LIN {X 0,Y 570.27,Z 1282.919,A -85,B 0,C 180,E1 9276.078,E2 9276.078} C_VEL
LIN {X 0,Y 570.578,Z 1274.301,A -85,B 0,C 180,E1 9280.677,E2 9280.677} C_VEL
LIN {X 0,Y 571.345,Z 1260.732,A -85,B 0,C 180,E1 9285.329,E2 9285.329} C_VEL
LIN {X 0,Y 573.008,Z 1241.765,A -85,B 0,C 180,E1 9290.042,E2 9290.042} C_VEL
LIN {X 0,Y 575.848,Z 1217.478,A -85,B 0,C 180,E1 9294.611,E2 9294.611} C_VEL
LIN {X 0,Y 580.222,Z 1187.751,A -85,B 0,C 180,E1 9299.027,E2 9299.027} C_VEL
LIN {X 0,Y 585.818,Z 1152.279,A -85,B 0,C 180,E1 9303.171,E2 9303.171} C_VEL
LIN {X 0,Y 592.121,Z 1114.219,A -85,B 0,C 180,E1 9306.711,E2 9306.711} C_VEL
LIN {X 0,Y 598.707,Z 1072.32,A -85,B 0,C 180,E1 9309.756,E2 9309.756} C_VEL
LIN {X 0,Y 603.11,Z 1037.935,A -85,B 0,C 180,E1 9311.685,E2 9311.685} C_VEL
LIN {X 0,Y 607.858,Z 987.119,A -85,B 0,C 180,E1 9313.723,E2 9313.723} C_VEL
LIN {X 0,Y 611.73,Z 933.476,A -85,B 0,C 180,E1 9315.186,E2 9315.186} C_VEL
LIN {X 0,Y 613.598,Z 886.911,A -85,B 0,C 180,E1 9315.996,E2 9315.996} C_VEL
LIN {X 0,Y 590.85,Z 850.721,A -85,B 0,C 180,E1 9318.163,E2 9318.163} C_VEL
LIN {X 0,Y 571.274,Z 814.347,A -85,B 0,C 180,E1 9320.427,E2 9320.427} C_VEL
LIN {X 0,Y 569.24,Z 809.06,A -85,B 0,C 180,E1 9320.777,E2 9320.777} C_VEL
LIN {X 0,Y 569.158,Z 809.06,A -85,B 0,C 180,E1 9326.116,E2 9326.116} C_VEL
LIN {X 0,Y 569.253,Z 809.06,A -85,B 0,C 180,E1 9331.459,E2 9331.459} C_VEL
LIN {X 0,Y 569.293,Z 809.111,A -85,B 0,C 180,E1 9336.25,E2 9336.25} C_VEL
LIN {X 0,Y 571.892,Z 814.911,A -85,B 0,C 180,E1 9336.731,E2 9336.731} C_VEL
LIN {X 0,Y 590.013,Z 852.89,A -85,B 0,C 180,E1 9340.042,E2 9340.042} C_VEL
LIN {X 0,Y 603.31,Z 886.116,A -85,B 0,C 180,E1 9343.049,E2 9343.049} C_VEL
LIN {X 0,Y 601.143,Z 906.53,A -85,B 0,C 180,E1 9344.23,E2 9344.23} C_VEL
LIN {X 0,Y 594.464,Z 949.147,A -85,B 0,C 180,E1 9347.056,E2 9347.056} C_VEL
LIN {X 0,Y 588.168,Z 988.3,A -85,B 0,C 180,E1 9350.387,E2 9350.387} C_VEL
LIN {X 0,Y 582.328,Z 1024.228,A -85,B 0,C 180,E1 9354.229,E2 9354.229} C_VEL
LIN {X 0,Y 577.319,Z 1057.198,A -85,B 0,C 180,E1 9358.687,E2 9358.687} C_VEL
LIN {X 0,Y 573.896,Z 1084.316,A -85,B 0,C 180,E1 9363.396,E2 9363.396} C_VEL
LIN {X 0,Y 571.748,Z 1105.972,A -85,B 0,C 180,E1 9368.299,E2 9368.299} C_VEL
LIN {X 0,Y 570.726,Z 1121.122,A -85,B 0,C 180,E1 9373.004,E2 9373.004} C_VEL
LIN {X 0,Y 570.222,Z 1130.776,A -85,B 0,C 180,E1 9377.472,E2 9377.472} C_VEL
LIN {X 0,Y 569.748,Z 1135.899,A -85,B 0,C 180,E1 9381.854,E2 9381.854} C_VEL
LIN {X 0,Y 569.684,Z 1136.615,A -85,B 0,C 180,E1 9386.801,E2 9386.801} C_VEL
LIN {X 0,Y 570.107,Z 1133.109,A -85,B 0,C 180,E1 9390.855,E2 9390.855} C_VEL
LIN {X 0,Y 570.541,Z 1124.317,A -85,B 0,C 180,E1 9395.635,E2 9395.635} C_VEL
LIN {X 0,Y 571.308,Z 1110.925,A -85,B 0,C 180,E1 9400.236,E2 9400.236} C_VEL
LIN {X 0,Y 572.975,Z 1091.952,A -85,B 0,C 180,E1 9404.949,E2 9404.949} C_VEL
LIN {X 0,Y 575.904,Z 1067.652,A -85,B 0,C 180,E1 9409.54,E2 9409.54} C_VEL
LIN {X 0,Y 580.109,Z 1037.955,A -85,B 0,C 180,E1 9413.951,E2 9413.951} C_VEL
LIN {X 0,Y 585.487,Z 1004.176,A -85,B 0,C 180,E1 9417.936,E2 9417.936} C_VEL
LIN {X 0,Y 591.862,Z 965.664,A -85,B 0,C 180,E1 9421.545,E2 9421.545} C_VEL
LIN {X 0,Y 598.661,Z 923.01,A -85,B 0,C 180,E1 9424.677,E2 9424.677} C_VEL
LIN {X 0,Y 603.556,Z 886.886,A -85,B 0,C 180,E1 9426.783,E2 9426.783} C_VEL
LIN {X 0,Y 589.393,Z 850.595,A -85,B 0,C 180,E1 9430.148,E2 9430.148} C_VEL
LIN {X 0,Y 571.501,Z 814.431,A -85,B 0,C 180,E1 9433.642,E2 9433.642} C_VEL
LIN {X 0,Y 569.436,Z 809.06,A -85,B 0,C 180,E1 9434.125,E2 9434.125} C_VEL
LIN {X 0,Y 569.824,Z 809.06,A -85,B 0,C 180,E1 9439.309,E2 9439.309} C_VEL
LIN {X 0,Y 570.01,Z 809.06,A -85,B 0,C 180,E1 9443.919,E2 9443.919} C_VEL
LIN {X 0,Y 570.065,Z 809.06,A -85,B 0,C 180,E1 9448.487,E2 9448.487} C_VEL
LIN {X 0,Y 570.001,Z 809.06,A -85,B 0,C 180,E1 9453.045,E2 9453.045} C_VEL
LIN {X 0,Y 569.951,Z 809.06,A -85,B 0,C 180,E1 9457.624,E2 9457.624} C_VEL
LIN {X 0,Y 569.806,Z 809.06,A -85,B 0,C 180,E1 9462.255,E2 9462.255} C_VEL
LIN {X 0,Y 569.672,Z 809.06,A -85,B 0,C 180,E1 9467.283,E2 9467.283} C_VEL
LIN {X 0,Y 569.54,Z 809.06,A -85,B 0,C 180,E1 9471.811,E2 9471.811} C_VEL
LIN {X 0,Y 569.423,Z 809.06,A -85,B 0,C 180,E1 9476.822,E2 9476.822} C_VEL
LIN {X 0,Y 569.313,Z 809.06,A -85,B 0,C 180,E1 9482.069,E2 9482.069} C_VEL
LIN {X 0,Y 569.252,Z 809.06,A -85,B 0,C 180,E1 9487.635,E2 9487.635} C_VEL
LIN {X 0,Y 569.19,Z 809.06,A -85,B 0,C 180,E1 9493.657,E2 9493.657} C_VEL
LIN {X 0,Y 569.157,Z 809.06,A -85,B 0,C 180,E1 9498.418,E2 9498.418} C_VEL
LIN {X 0,Y 569.22,Z 809.06,A -85,B 0,C 180,E1 9504.269,E2 9504.269} C_VEL
LIN {X 0,Y 569.324,Z 809.06,A -85,B 0,C 180,E1 9509.718,E2 9509.718} C_VEL
LIN {X 0,Y 569.49,Z 809.06,A -85,B 0,C 180,E1 9514.881,E2 9514.881} C_VEL
LIN {X 0,Y 569.623,Z 809.06,A -85,B 0,C 180,E1 9519.829,E2 9519.829} C_VEL
LIN {X 0,Y 569.678,Z 809.06,A -85,B 0,C 180,E1 9524.62,E2 9524.62} C_VEL
LIN {X 0,Y 569.836,Z 809.06,A -85,B 0,C 180,E1 9529.304,E2 9529.304} C_VEL
LIN {X 0,Y 570.009,Z 809.06,A -85,B 0,C 180,E1 9533.914,E2 9533.914} C_VEL
LIN {X 0,Y 570.293,Z 809.06,A -85,B 0,C 180,E1 9540.001,E2 9540.001} C_VEL
LIN {X 0,Y 570.05,Z 809.06,A -85,B 0,C 180,E1 9546.087,E2 9546.087} C_VEL
LIN {X 0,Y 569.806,Z 809.06,A -85,B 0,C 180,E1 9552.248,E2 9552.248} C_VEL
LIN {X 0,Y 569.663,Z 809.06,A -85,B 0,C 180,E1 9557.251,E2 9557.251} C_VEL
LIN {X 0,Y 569.537,Z 809.06,A -85,B 0,C 180,E1 9561.804,E2 9561.804} C_VEL
LIN {X 0,Y 569.373,Z 809.06,A -85,B 0,C 180,E1 9566.818,E2 9566.818} C_VEL
LIN {X 0,Y 569.312,Z 809.06,A -85,B 0,C 180,E1 9572.061,E2 9572.061} C_VEL
LIN {X 0,Y 569.281,Z 809.538,A -85,B 0,C 180,E1 9577.816,E2 9577.816} C_VEL
LIN {X 0,Y 571.948,Z 814.98,A -85,B 0,C 180,E1 9578.222,E2 9578.222} C_VEL
LIN {X 0,Y 598.675,Z 858.988,A -85,B 0,C 180,E1 9581.795,E2 9581.795} C_VEL
LIN {X 0,Y 615.701,Z 888.66,A -85,B 0,C 180,E1 9583.807,E2 9583.807} C_VEL
LIN {X 0,Y 613.152,Z 939.54,A -85,B 0,C 180,E1 9584.758,E2 9584.758} C_VEL
LIN {X 0,Y 609.127,Z 984.504,A -85,B 0,C 180,E1 9586.049,E2 9586.049} C_VEL
LIN {X 0,Y 604.919,Z 1025.197,A -85,B 0,C 180,E1 9587.692,E2 9587.692} C_VEL
LIN {X 0,Y 599.652,Z 1040.997,A -85,B 0,C 180,E1 9588.224,E2 9588.224} C_VEL
LIN {X 0,Y 594.647,Z 1054.535,A -85,B 0,C 180,E1 9588.734,E2 9588.734} C_VEL
LIN {X 0,Y 594.367,Z 1056.402,A -85,B 0,C 180,E1 9588.836,E2 9588.836} C_VEL
LIN {X 0,Y 589.081,Z 1093.061,A -85,B 0,C 180,E1 9591.166,E2 9591.166} C_VEL
LIN {X 0,Y 582.379,Z 1132.494,A -85,B 0,C 180,E1 9594.416,E2 9594.416} C_VEL
LIN {X 0,Y 575.672,Z 1171.448,A -85,B 0,C 180,E1 9598.523,E2 9598.523} C_VEL
LIN {X 0,Y 570.444,Z 1203.465,A -85,B 0,C 180,E1 9602.806,E2 9602.806} C_VEL
LIN {X 0,Y 566.697,Z 1230.555,A -85,B 0,C 180,E1 9607.393,E2 9607.393} C_VEL
LIN {X 0,Y 564.414,Z 1251.77,A -85,B 0,C 180,E1 9612.025,E2 9612.025} C_VEL
LIN {X 0,Y 562.989,Z 1268.116,A -85,B 0,C 180,E1 9616.806,E2 9616.806} C_VEL
LIN {X 0,Y 562.467,Z 1279.21,A -85,B 0,C 180,E1 9621.497,E2 9621.497} C_VEL
LIN {X 0,Y 562.279,Z 1284.659,A -85,B 0,C 180,E1 9625.369,E2 9625.369} C_VEL
LIN {X 0,Y 562.346,Z 1287,A -85,B 0,C 180,E1 9629.994,E2 9629.994} C_VEL
LIN {X 0,Y 562.279,Z 1284.673,A -85,B 0,C 180,E1 9634.618,E2 9634.618} C_VEL
LIN {X 0,Y 562.448,Z 1277.69,A -85,B 0,C 180,E1 9639.27,E2 9639.27} C_VEL
LIN {X 0,Y 563.222,Z 1265.86,A -85,B 0,C 180,E1 9643.966,E2 9643.966} C_VEL
LIN {X 0,Y 564.723,Z 1248.729,A -85,B 0,C 180,E1 9648.722,E2 9648.722} C_VEL
LIN {X 0,Y 567.547,Z 1224.45,A -85,B 0,C 180,E1 9653.74,E2 9653.74} C_VEL
LIN {X 0,Y 571.579,Z 1196.601,A -85,B 0,C 180,E1 9658.197,E2 9658.197} C_VEL
LIN {X 0,Y 577.41,Z 1161.259,A -85,B 0,C 180,E1 9662.659,E2 9662.659} C_VEL
LIN {X 0,Y 583.923,Z 1123.342,A -85,B 0,C 180,E1 9666.403,E2 9666.403} C_VEL
LIN {X 0,Y 590.741,Z 1082.843,A -85,B 0,C 180,E1 9669.569,E2 9669.569} C_VEL
LIN {X 0,Y 595.524,Z 1043.572,A -85,B 0,C 180,E1 9671.766,E2 9671.766} C_VEL
LIN {X 0,Y 600.653,Z 991.518,A -85,B 0,C 180,E1 9673.943,E2 9673.943} C_VEL
LIN {X 0,Y 604.673,Z 940.832,A -85,B 0,C 180,E1 9675.437,E2 9675.437} C_VEL
LIN {X 0,Y 607.027,Z 889.973,A -85,B 0,C 180,E1 9676.388,E2 9676.388} C_VEL
LIN {X 0,Y 585.603,Z 855.505,A -85,B 0,C 180,E1 9678.501,E2 9678.501} C_VEL
LIN {X 0,Y 566.705,Z 819.88,A -85,B 0,C 180,E1 9680.764,E2 9680.764} C_VEL
LIN {X 0,Y 561.456,Z 810.557,A -85,B 0,C 180,E1 9681.473,E2 9681.473} C_VEL
LIN {X 0,Y 561.314,Z 809.06,A -85,B 0,C 180,E1 9681.557,E2 9681.557} C_VEL
LIN {X 0,Y 561.235,Z 809.06,A -85,B 0,C 180,E1 9687.421,E2 9687.421} C_VEL
LIN {X 0,Y 561.342,Z 809.06,A -85,B 0,C 180,E1 9692.767,E2 9692.767} C_VEL
LIN {X 0,Y 561.39,Z 809.624,A -85,B 0,C 180,E1 9695.4,E2 9695.4} C_VEL
LIN {X 0,Y 567.085,Z 820.612,A -85,B 0,C 180,E1 9696.428,E2 9696.428} C_VEL
LIN {X 0,Y 584.99,Z 858.969,A -85,B 0,C 180,E1 9699.894,E2 9699.894} C_VEL
LIN {X 0,Y 597.178,Z 890.245,A -85,B 0,C 180,E1 9702.783,E2 9702.783} C_VEL
LIN {X 0,Y 590.812,Z 932.783,A -85,B 0,C 180,E1 9705.371,E2 9705.371} C_VEL
LIN {X 0,Y 583.573,Z 975.191,A -85,B 0,C 180,E1 9708.707,E2 9708.707} C_VEL
LIN {X 0,Y 577.139,Z 1012.847,A -85,B 0,C 180,E1 9712.478,E2 9712.478} C_VEL
LIN {X 0,Y 571.505,Z 1046.855,A -85,B 0,C 180,E1 9716.779,E2 9716.779} C_VEL
LIN {X 0,Y 567.399,Z 1075.144,A -85,B 0,C 180,E1 9721.335,E2 9721.335} C_VEL
LIN {X 0,Y 564.565,Z 1098.396,A -85,B 0,C 180,E1 9726.145,E2 9726.145} C_VEL
LIN {X 0,Y 563.206,Z 1115.371,A -85,B 0,C 180,E1 9730.824,E2 9730.824} C_VEL
LIN {X 0,Y 562.453,Z 1127.522,A -85,B 0,C 180,E1 9735.583,E2 9735.583} C_VEL
LIN {X 0,Y 562.058,Z 1134.141,A -85,B 0,C 180,E1 9739.808,E2 9739.808} C_VEL
LIN {X 0,Y 561.734,Z 1136.813,A -85,B 0,C 180,E1 9743.868,E2 9743.868} C_VEL
LIN {X 0,Y 561.918,Z 1135.246,A -85,B 0,C 180,E1 9748.947,E2 9748.947} C_VEL
LIN {X 0,Y 562.493,Z 1128.891,A -85,B 0,C 180,E1 9753.628,E2 9753.628} C_VEL
LIN {X 0,Y 563.215,Z 1117.089,A -85,B 0,C 180,E1 9758.519,E2 9758.519} C_VEL
LIN {X 0,Y 564.477,Z 1099.987,A -85,B 0,C 180,E1 9763.383,E2 9763.383} C_VEL
LIN {X 0,Y 566.914,Z 1078.804,A -85,B 0,C 180,E1 9767.898,E2 9767.898} C_VEL
LIN {X 0,Y 570.861,Z 1050.717,A -85,B 0,C 180,E1 9772.565,E2 9772.565} C_VEL
LIN {X 0,Y 576.205,Z 1017.971,A -85,B 0,C 180,E1 9776.844,E2 9776.844} C_VEL
LIN {X 0,Y 582.483,Z 981.653,A -85,B 0,C 180,E1 9780.615,E2 9780.615} C_VEL
LIN {X 0,Y 589.351,Z 941.758,A -85,B 0,C 180,E1 9783.889,E2 9783.889} C_VEL
LIN {X 0,Y 595.881,Z 900.345,A -85,B 0,C 180,E1 9786.563,E2 9786.563} C_VEL
LIN {X 0,Y 597.083,Z 889.866,A -85,B 0,C 180,E1 9787.156,E2 9787.156} C_VEL
LIN {X 0,Y 583.392,Z 854.423,A -85,B 0,C 180,E1 9790.527,E2 9790.527} C_VEL
LIN {X 0,Y 566.082,Z 819.268,A -85,B 0,C 180,E1 9794.026,E2 9794.026} C_VEL
LIN {X 0,Y 561.565,Z 809.06,A -85,B 0,C 180,E1 9795.024,E2 9795.024} C_VEL
LIN {X 0,Y 561.986,Z 809.06,A -85,B 0,C 180,E1 9800.723,E2 9800.723} C_VEL
LIN {X 0,Y 562.129,Z 809.06,A -85,B 0,C 180,E1 9805.381,E2 9805.381} C_VEL
LIN {X 0,Y 562.245,Z 809.06,A -85,B 0,C 180,E1 9811.546,E2 9811.546} C_VEL
LIN {X 0,Y 562.11,Z 809.06,A -85,B 0,C 180,E1 9816.179,E2 9816.179} C_VEL
LIN {X 0,Y 561.94,Z 809.06,A -85,B 0,C 180,E1 9820.856,E2 9820.856} C_VEL
LIN {X 0,Y 561.813,Z 809.06,A -85,B 0,C 180,E1 9825.609,E2 9825.609} C_VEL
LIN {X 0,Y 561.669,Z 809.06,A -85,B 0,C 180,E1 9830.478,E2 9830.478} C_VEL
LIN {X 0,Y 561.519,Z 809.06,A -85,B 0,C 180,E1 9835.51,E2 9835.51} C_VEL
LIN {X 0,Y 561.41,Z 809.06,A -85,B 0,C 180,E1 9840.764,E2 9840.764} C_VEL
LIN {X 0,Y 561.34,Z 809.06,A -85,B 0,C 180,E1 9846.322,E2 9846.322} C_VEL
LIN {X 0,Y 561.249,Z 809.06,A -85,B 0,C 180,E1 9852.313,E2 9852.313} C_VEL
LIN {X 0,Y 561.215,Z 809.06,A -85,B 0,C 180,E1 9857.695,E2 9857.695} C_VEL
LIN {X 0,Y 561.288,Z 809.06,A -85,B 0,C 180,E1 9863.876,E2 9863.876} C_VEL
LIN {X 0,Y 561.394,Z 809.06,A -85,B 0,C 180,E1 9869.476,E2 9869.476} C_VEL
LIN {X 0,Y 561.589,Z 809.06,A -85,B 0,C 180,E1 9874.502,E2 9874.502} C_VEL
LIN {X 0,Y 561.707,Z 809.06,A -85,B 0,C 180,E1 9880.329,E2 9880.329} C_VEL
LIN {X 0,Y 561.779,Z 809.06,A -85,B 0,C 180,E1 9885.992,E2 9885.992} C_VEL
LIN {X 0,Y 562.015,Z 809.06,A -85,B 0,C 180,E1 9890.718,E2 9890.718} C_VEL
LIN {X 0,Y 562.162,Z 809.06,A -85,B 0,C 180,E1 9895.376,E2 9895.376} C_VEL
LIN {X 0,Y 562.382,Z 809.06,A -85,B 0,C 180,E1 9901.54,E2 9901.54} C_VEL
LIN {X 0,Y 562.143,Z 809.06,A -85,B 0,C 180,E1 9906.173,E2 9906.173} C_VEL
LIN {X 0,Y 561.943,Z 809.06,A -85,B 0,C 180,E1 9910.85,E2 9910.85} C_VEL
LIN {X 0,Y 561.789,Z 809.06,A -85,B 0,C 180,E1 9915.603,E2 9915.603} C_VEL
LIN {X 0,Y 561.66,Z 809.06,A -85,B 0,C 180,E1 9920.471,E2 9920.471} C_VEL
LIN {X 0,Y 561.494,Z 809.06,A -85,B 0,C 180,E1 9925.504,E2 9925.504} C_VEL
LIN {X 0,Y 561.401,Z 809.06,A -85,B 0,C 180,E1 9930.756,E2 9930.756} C_VEL
LIN {X 0,Y 561.363,Z 809.06,A -85,B 0,C 180,E1 9936.9,E2 9936.9} C_VEL
LIN {X 0,Y 563.774,Z 814.722,A -85,B 0,C 180,E1 9937.305,E2 9937.305} C_VEL
LIN {X 0,Y 591.925,Z 860.297,A -85,B 0,C 180,E1 9941.157,E2 9941.157} C_VEL
LIN {X 0,Y 609.778,Z 892.169,A -85,B 0,C 180,E1 9943.358,E2 9943.358} C_VEL
LIN {X 0,Y 606.664,Z 945.689,A -85,B 0,C 180,E1 9944.411,E2 9944.411} C_VEL
LIN {X 0,Y 602.242,Z 991.336,A -85,B 0,C 180,E1 9945.821,E2 9945.821} C_VEL
LIN {X 0,Y 596.519,Z 1040.194,A -85,B 0,C 180,E1 9947.969,E2 9947.969} C_VEL
LIN {X 0,Y 594.367,Z 1056.402,A -85,B 0,C 180,E1 9948.836,E2 9948.836} C_VEL
LIN {X 0,Y 590.876,Z 1067.886,A -85,B 0,C 180,E1 9949.369,E2 9949.369} C_VEL
LIN {X 0,Y 583.812,Z 1084.601,A -85,B 0,C 180,E1 9950.139,E2 9950.139} C_VEL
LIN {X 0,Y 583.429,Z 1086.38,A -85,B 0,C 180,E1 9950.256,E2 9950.256} C_VEL
LIN {X 0,Y 577.779,Z 1120.685,A -85,B 0,C 180,E1 9952.876,E2 9952.876} C_VEL
LIN {X 0,Y 570.593,Z 1160.391,A -85,B 0,C 180,E1 9956.791,E2 9956.791} C_VEL
LIN {X 0,Y 564.417,Z 1195.079,A -85,B 0,C 180,E1 9961.184,E2 9961.184} C_VEL
LIN {X 0,Y 560.043,Z 1223.282,A -85,B 0,C 180,E1 9965.697,E2 9965.697} C_VEL
LIN {X 0,Y 557.015,Z 1246.941,A -85,B 0,C 180,E1 9970.584,E2 9970.584} C_VEL
LIN {X 0,Y 555.479,Z 1264.335,A -85,B 0,C 180,E1 9975.314,E2 9975.314} C_VEL
LIN {X 0,Y 554.708,Z 1276.093,A -85,B 0,C 180,E1 9979.795,E2 9979.795} C_VEL
LIN {X 0,Y 554.545,Z 1282.902,A -85,B 0,C 180,E1 9983.736,E2 9983.736} C_VEL
LIN {X 0,Y 554.354,Z 1286.665,A -85,B 0,C 180,E1 9988.432,E2 9988.432} C_VEL
LIN {X 0,Y 554.494,Z 1285.879,A -85,B 0,C 180,E1 9993.118,E2 9993.118} C_VEL
LIN {X 0,Y 554.505,Z 1280.558,A -85,B 0,C 180,E1 9997.825,E2 9997.825} C_VEL
LIN {X 0,Y 555.052,Z 1270.437,A -85,B 0,C 180,E1 10002.573,E2 10002.573} C_VEL
LIN {X 0,Y 556.257,Z 1255.027,A -85,B 0,C 180,E1 10007.379,E2 10007.379} C_VEL
LIN {X 0,Y 558.828,Z 1232.701,A -85,B 0,C 180,E1 10012.516,E2 10012.516} C_VEL
LIN {X 0,Y 562.749,Z 1206.183,A -85,B 0,C 180,E1 10017.152,E2 10017.152} C_VEL
LIN {X 0,Y 568.149,Z 1174.436,A -85,B 0,C 180,E1 10021.556,E2 10021.556} C_VEL
LIN {X 0,Y 574.679,Z 1137.631,A -85,B 0,C 180,E1 10025.566,E2 10025.566} C_VEL
LIN {X 0,Y 581.17,Z 1100.835,A -85,B 0,C 180,E1 10028.741,E2 10028.741} C_VEL
LIN {X 0,Y 586.709,Z 1058.959,A -85,B 0,C 180,E1 10031.311,E2 10031.311} C_VEL
LIN {X 0,Y 592.045,Z 1011.546,A -85,B 0,C 180,E1 10033.551,E2 10033.551} C_VEL
LIN {X 0,Y 596.302,Z 965.395,A -85,B 0,C 180,E1 10035.188,E2 10035.188} C_VEL
LIN {X 0,Y 599.852,Z 915.853,A -85,B 0,C 180,E1 10036.375,E2 10036.375} C_VEL
LIN {X 0,Y 600.289,Z 892.715,A -85,B 0,C 180,E1 10036.808,E2 10036.808} C_VEL
LIN {X 0,Y 580.66,Z 860.751,A -85,B 0,C 180,E1 10038.818,E2 10038.818} C_VEL
LIN {X 0,Y 561.82,Z 824.949,A -85,B 0,C 180,E1 10041.155,E2 10041.155} C_VEL
LIN {X 0,Y 553.395,Z 809.959,A -85,B 0,C 180,E1 10042.379,E2 10042.379} C_VEL
LIN {X 0,Y 553.322,Z 809.06,A -85,B 0,C 180,E1 10042.664,E2 10042.664} C_VEL
LIN {X 0,Y 553.335,Z 809.06,A -85,B 0,C 180,E1 10048.745,E2 10048.745} C_VEL
LIN {X 0,Y 553.505,Z 809.41,A -85,B 0,C 180,E1 10054.458,E2 10054.458} C_VEL
LIN {X 0,Y 556.013,Z 814.843,A -85,B 0,C 180,E1 10054.944,E2 10054.944} C_VEL
LIN {X 0,Y 572.142,Z 846.836,A -85,B 0,C 180,E1 10058.053,E2 10058.053} C_VEL
LIN {X 0,Y 588.015,Z 885.193,A -85,B 0,C 180,E1 10061.64,E2 10061.64} C_VEL
LIN {X 0,Y 590.789,Z 895.257,A -85,B 0,C 180,E1 10062.545,E2 10062.545} C_VEL
LIN {X 0,Y 584.32,Z 935.414,A -85,B 0,C 180,E1 10065.013,E2 10065.013} C_VEL
LIN {X 0,Y 576.622,Z 976.931,A -85,B 0,C 180,E1 10068.378,E2 10068.378} C_VEL
LIN {X 0,Y 569.917,Z 1014.273,A -85,B 0,C 180,E1 10072.19,E2 10072.19} C_VEL
LIN {X 0,Y 564.035,Z 1047.94,A -85,B 0,C 180,E1 10076.544,E2 10076.544} C_VEL
LIN {X 0,Y 559.732,Z 1076.008,A -85,B 0,C 180,E1 10081.16,E2 10081.16} C_VEL
LIN {X 0,Y 556.861,Z 1098.253,A -85,B 0,C 180,E1 10085.84,E2 10085.84} C_VEL
LIN {X 0,Y 555.383,Z 1115.255,A -85,B 0,C 180,E1 10090.581,E2 10090.581} C_VEL
LIN {X 0,Y 554.621,Z 1126.648,A -85,B 0,C 180,E1 10095.007,E2 10095.007} C_VEL
LIN {X 0,Y 554.269,Z 1133.364,A -85,B 0,C 180,E1 10099.094,E2 10099.094} C_VEL
LIN {X 0,Y 553.879,Z 1136.295,A -85,B 0,C 180,E1 10102.452,E2 10102.452} C_VEL
LIN {X 0,Y 553.875,Z 1136.202,A -85,B 0,C 180,E1 10107.63,E2 10107.63} C_VEL
LIN {X 0,Y 554.431,Z 1131.238,A -85,B 0,C 180,E1 10112.354,E2 10112.354} C_VEL
LIN {X 0,Y 554.941,Z 1122.283,A -85,B 0,C 180,E1 10116.799,E2 10116.799} C_VEL
LIN {X 0,Y 556.067,Z 1107.32,A -85,B 0,C 180,E1 10121.734,E2 10121.734} C_VEL
LIN {X 0,Y 558.561,Z 1085.383,A -85,B 0,C 180,E1 10126.918,E2 10126.918} C_VEL
LIN {X 0,Y 562.225,Z 1059.784,A -85,B 0,C 180,E1 10131.546,E2 10131.546} C_VEL
LIN {X 0,Y 567.33,Z 1028.5,A -85,B 0,C 180,E1 10135.999,E2 10135.999} C_VEL
LIN {X 0,Y 573.689,Z 993.193,A -85,B 0,C 180,E1 10139.978,E2 10139.978} C_VEL
LIN {X 0,Y 581.167,Z 952.357,A -85,B 0,C 180,E1 10143.61,E2 10143.61} C_VEL
LIN {X 0,Y 588.328,Z 909.971,A -85,B 0,C 180,E1 10146.541,E2 10146.541} C_VEL
LIN {X 0,Y 590.888,Z 893.797,A -85,B 0,C 180,E1 10147.45,E2 10147.45} C_VEL
LIN {X 0,Y 577.472,Z 858.329,A -85,B 0,C 180,E1 10150.903,E2 10150.903} C_VEL
LIN {X 0,Y 559.287,Z 820.62,A -85,B 0,C 180,E1 10154.734,E2 10154.734} C_VEL
LIN {X 0,Y 553.858,Z 810.471,A -85,B 0,C 180,E1 10155.793,E2 10155.793} C_VEL
LIN {X 0,Y 553.777,Z 809.06,A -85,B 0,C 180,E1 10155.992,E2 10155.992} C_VEL
LIN {X 0,Y 554.063,Z 809.06,A -85,B 0,C 180,E1 10160.589,E2 10160.589} C_VEL
LIN {X 0,Y 554.252,Z 809.06,A -85,B 0,C 180,E1 10165.315,E2 10165.315} C_VEL
LIN {X 0,Y 554.346,Z 809.06,A -85,B 0,C 180,E1 10171.568,E2 10171.568} C_VEL
LIN {X 0,Y 554.195,Z 809.06,A -85,B 0,C 180,E1 10176.268,E2 10176.268} C_VEL
LIN {X 0,Y 554.027,Z 809.06,A -85,B 0,C 180,E1 10181.013,E2 10181.013} C_VEL
LIN {X 0,Y 553.884,Z 809.06,A -85,B 0,C 180,E1 10185.838,E2 10185.838} C_VEL
LIN {X 0,Y 553.719,Z 809.06,A -85,B 0,C 180,E1 10190.785,E2 10190.785} C_VEL
LIN {X 0,Y 553.572,Z 809.06,A -85,B 0,C 180,E1 10195.903,E2 10195.903} C_VEL
LIN {X 0,Y 553.436,Z 809.06,A -85,B 0,C 180,E1 10201.256,E2 10201.256} C_VEL
LIN {X 0,Y 553.346,Z 809.06,A -85,B 0,C 180,E1 10206.933,E2 10206.933} C_VEL
LIN {X 0,Y 553.361,Z 809.06,A -85,B 0,C 180,E1 10213.061,E2 10213.061} C_VEL
LIN {X 0,Y 553.29,Z 809.06,A -85,B 0,C 180,E1 10219.049,E2 10219.049} C_VEL
LIN {X 0,Y 553.348,Z 809.06,A -85,B 0,C 180,E1 10225.018,E2 10225.018} C_VEL
LIN {X 0,Y 553.55,Z 809.06,A -85,B 0,C 180,E1 10230.883,E2 10230.883} C_VEL
LIN {X 0,Y 553.643,Z 809.06,A -85,B 0,C 180,E1 10235.835,E2 10235.835} C_VEL
LIN {X 0,Y 553.835,Z 809.06,A -85,B 0,C 180,E1 10240.89,E2 10240.89} C_VEL
LIN {X 0,Y 553.883,Z 809.06,A -85,B 0,C 180,E1 10245.788,E2 10245.788} C_VEL
LIN {X 0,Y 554.091,Z 809.06,A -85,B 0,C 180,E1 10250.584,E2 10250.584} C_VEL
LIN {X 0,Y 554.262,Z 809.06,A -85,B 0,C 180,E1 10255.309,E2 10255.309} C_VEL
LIN {X 0,Y 554.478,Z 809.06,A -85,B 0,C 180,E1 10261.562,E2 10261.562} C_VEL
LIN {X 0,Y 554.227,Z 809.06,A -85,B 0,C 180,E1 10266.261,E2 10266.261} C_VEL
LIN {X 0,Y 554.021,Z 809.06,A -85,B 0,C 180,E1 10271.007,E2 10271.007} C_VEL
LIN {X 0,Y 553.861,Z 809.06,A -85,B 0,C 180,E1 10277.258,E2 10277.258} C_VEL
LIN {X 0,Y 553.63,Z 809.06,A -85,B 0,C 180,E1 10282.464,E2 10282.464} C_VEL
LIN {X 0,Y 553.504,Z 809.06,A -85,B 0,C 180,E1 10287.651,E2 10287.651} C_VEL
LIN {X 0,Y 553.421,Z 809.06,A -85,B 0,C 180,E1 10293.097,E2 10293.097} C_VEL
LIN {X 0,Y 553.462,Z 809.06,A -85,B 0,C 180,E1 10295.952,E2 10295.952} C_VEL
LIN {X 0,Y 555.857,Z 814.736,A -85,B 0,C 180,E1 10296.375,E2 10296.375} C_VEL
LIN {X 0,Y 585.368,Z 861.947,A -85,B 0,C 180,E1 10300.526,E2 10300.526} C_VEL
LIN {X 0,Y 603.778,Z 894.099,A -85,B 0,C 180,E1 10302.863,E2 10302.863} C_VEL
LIN {X 0,Y 600.627,Z 946.855,A -85,B 0,C 180,E1 10303.942,E2 10303.942} C_VEL
LIN {X 0,Y 595.992,Z 991.688,A -85,B 0,C 180,E1 10305.357,E2 10305.357} C_VEL
LIN {X 0,Y 589.933,Z 1040.905,A -85,B 0,C 180,E1 10307.552,E2 10307.552} C_VEL
LIN {X 0,Y 583.429,Z 1086.38,A -85,B 0,C 180,E1 10310.256,E2 10310.256} C_VEL
LIN {X 0,Y 577.747,Z 1100.839,A -85,B 0,C 180,E1 10311.06,E2 10311.06} C_VEL
LIN {X 0,Y 572.077,Z 1114.879,A -85,B 0,C 180,E1 10311.934,E2 10311.934} C_VEL
LIN {X 0,Y 566.629,Z 1145.24,A -85,B 0,C 180,E1 10314.703,E2 10314.703} C_VEL
LIN {X 0,Y 559.854,Z 1180.913,A -85,B 0,C 180,E1 10318.84,E2 10318.84} C_VEL
LIN {X 0,Y 554.546,Z 1211.371,A -85,B 0,C 180,E1 10323.275,E2 10323.275} C_VEL
LIN {X 0,Y 550.48,Z 1237.847,A -85,B 0,C 180,E1 10328.242,E2 10328.242} C_VEL
LIN {X 0,Y 548.2,Z 1257.996,A -85,B 0,C 180,E1 10333.17,E2 10333.17} C_VEL
LIN {X 0,Y 546.996,Z 1272.347,A -85,B 0,C 180,E1 10338.036,E2 10338.036} C_VEL
LIN {X 0,Y 546.644,Z 1281.741,A -85,B 0,C 180,E1 10342.848,E2 10342.848} C_VEL
LIN {X 0,Y 546.536,Z 1285.87,A -85,B 0,C 180,E1 10346.824,E2 10346.824} C_VEL
LIN {X 0,Y 546.696,Z 1286.668,A -85,B 0,C 180,E1 10351.577,E2 10351.577} C_VEL
LIN {X 0,Y 546.621,Z 1282.919,A -85,B 0,C 180,E1 10356.342,E2 10356.342} C_VEL
LIN {X 0,Y 547.007,Z 1274.3,A -85,B 0,C 180,E1 10361.143,E2 10361.143} C_VEL
LIN {X 0,Y 547.884,Z 1260.729,A -85,B 0,C 180,E1 10366.003,E2 10366.003} C_VEL
LIN {X 0,Y 549.994,Z 1241.769,A -85,B 0,C 180,E1 10370.919,E2 10370.919} C_VEL
LIN {X 0,Y 553.443,Z 1217.269,A -85,B 0,C 180,E1 10375.715,E2 10375.715} C_VEL
LIN {X 0,Y 558.719,Z 1187.081,A -85,B 0,C 180,E1 10380.359,E2 10380.359} C_VEL
LIN {X 0,Y 565.547,Z 1150.517,A -85,B 0,C 180,E1 10384.738,E2 10384.738} C_VEL
LIN {X 0,Y 571.289,Z 1119.314,A -85,B 0,C 180,E1 10387.694,E2 10387.694} C_VEL
LIN {X 0,Y 577.242,Z 1077.007,A -85,B 0,C 180,E1 10390.614,E2 10390.614} C_VEL
LIN {X 0,Y 583.249,Z 1028.297,A -85,B 0,C 180,E1 10393.204,E2 10393.204} C_VEL
LIN {X 0,Y 588.336,Z 978.716,A -85,B 0,C 180,E1 10395.179,E2 10395.179} C_VEL
LIN {X 0,Y 592.758,Z 924.306,A -85,B 0,C 180,E1 10396.648,E2 10396.648} C_VEL
LIN {X 0,Y 594.083,Z 896.271,A -85,B 0,C 180,E1 10397.19,E2 10397.19} C_VEL
LIN {X 0,Y 575.538,Z 865.659,A -85,B 0,C 180,E1 10399.165,E2 10399.165} C_VEL
LIN {X 0,Y 557.41,Z 830.55,A -85,B 0,C 180,E1 10401.502,E2 10401.502} C_VEL
LIN {X 0,Y 547.425,Z 814.299,A -85,B 0,C 180,E1 10403.009,E2 10403.009} C_VEL
LIN {X 0,Y 545.384,Z 809.06,A -85,B 0,C 180,E1 10403.452,E2 10403.452} C_VEL
LIN {X 0,Y 545.404,Z 809.06,A -85,B 0,C 180,E1 10409.176,E2 10409.176} C_VEL
LIN {X 0,Y 545.478,Z 809.081,A -85,B 0,C 180,E1 10413.369,E2 10413.369} C_VEL
LIN {X 0,Y 547.858,Z 814.678,A -85,B 0,C 180,E1 10413.907,E2 10413.907} C_VEL
LIN {X 0,Y 562.413,Z 841.845,A -85,B 0,C 180,E1 10416.794,E2 10416.794} C_VEL
LIN {X 0,Y 579.201,Z 881.834,A -85,B 0,C 180,E1 10420.63,E2 10420.63} C_VEL
LIN {X 0,Y 584.454,Z 898.006,A -85,B 0,C 180,E1 10422.155,E2 10422.155} C_VEL
LIN {X 0,Y 577.836,Z 938.057,A -85,B 0,C 180,E1 10424.647,E2 10424.647} C_VEL
LIN {X 0,Y 570.352,Z 975.968,A -85,B 0,C 180,E1 10427.763,E2 10427.763} C_VEL
LIN {X 0,Y 562.437,Z 1017.234,A -85,B 0,C 180,E1 10432.086,E2 10432.086} C_VEL
LIN {X 0,Y 556.309,Z 1050.31,A -85,B 0,C 180,E1 10436.496,E2 10436.496} C_VEL
LIN {X 0,Y 551.94,Z 1077.668,A -85,B 0,C 180,E1 10441.132,E2 10441.132} C_VEL
LIN {X 0,Y 548.993,Z 1099.711,A -85,B 0,C 180,E1 10445.924,E2 10445.924} C_VEL
LIN {X 0,Y 547.486,Z 1116.323,A -85,B 0,C 180,E1 10450.736,E2 10450.736} C_VEL
LIN {X 0,Y 546.706,Z 1127.418,A -85,B 0,C 180,E1 10455.257,E2 10455.257} C_VEL
LIN {X 0,Y 546.221,Z 1134.381,A -85,B 0,C 180,E1 10459.873,E2 10459.873} C_VEL
LIN {X 0,Y 545.885,Z 1136.932,A -85,B 0,C 180,E1 10464.531,E2 10464.531} C_VEL
LIN {X 0,Y 545.992,Z 1135.986,A -85,B 0,C 180,E1 10468.064,E2 10468.064} C_VEL
LIN {X 0,Y 546.579,Z 1130.587,A -85,B 0,C 180,E1 10472.877,E2 10472.877} C_VEL
LIN {X 0,Y 547.175,Z 1121.173,A -85,B 0,C 180,E1 10477.409,E2 10477.409} C_VEL
LIN {X 0,Y 548.389,Z 1106.254,A -85,B 0,C 180,E1 10482.266,E2 10482.266} C_VEL
LIN {X 0,Y 550.908,Z 1085.696,A -85,B 0,C 180,E1 10487.174,E2 10487.174} C_VEL
LIN {X 0,Y 554.841,Z 1059.535,A -85,B 0,C 180,E1 10491.97,E2 10491.97} C_VEL
LIN {X 0,Y 560.258,Z 1028.432,A -85,B 0,C 180,E1 10496.444,E2 10496.444} C_VEL
LIN {X 0,Y 566.799,Z 993.853,A -85,B 0,C 180,E1 10500.391,E2 10500.391} C_VEL
LIN {X 0,Y 574.631,Z 953.868,A -85,B 0,C 180,E1 10504.025,E2 10504.025} C_VEL
LIN {X 0,Y 582.028,Z 911.877,A -85,B 0,C 180,E1 10506.965,E2 10506.965} C_VEL
LIN {X 0,Y 584.304,Z 896.295,A -85,B 0,C 180,E1 10507.884,E2 10507.884} C_VEL
LIN {X 0,Y 570.73,Z 860.32,A -85,B 0,C 180,E1 10511.482,E2 10511.482} C_VEL
LIN {X 0,Y 553.427,Z 824.69,A -85,B 0,C 180,E1 10515.226,E2 10515.226} C_VEL
LIN {X 0,Y 545.944,Z 809.959,A -85,B 0,C 180,E1 10516.756,E2 10516.756} C_VEL
LIN {X 0,Y 545.944,Z 809.06,A -85,B 0,C 180,E1 10517.214,E2 10517.214} C_VEL
LIN {X 0,Y 546.239,Z 809.06,A -85,B 0,C 180,E1 10522.056,E2 10522.056} C_VEL
LIN {X 0,Y 546.414,Z 809.06,A -85,B 0,C 180,E1 10526.836,E2 10526.836} C_VEL
LIN {X 0,Y 546.44,Z 809.06,A -85,B 0,C 180,E1 10531.591,E2 10531.591} C_VEL
LIN {X 0,Y 546.31,Z 809.06,A -85,B 0,C 180,E1 10536.359,E2 10536.359} C_VEL
LIN {X 0,Y 546.102,Z 809.06,A -85,B 0,C 180,E1 10541.175,E2 10541.175} C_VEL
LIN {X 0,Y 545.963,Z 809.06,A -85,B 0,C 180,E1 10546.074,E2 10546.074} C_VEL
LIN {X 0,Y 545.789,Z 809.06,A -85,B 0,C 180,E1 10551.102,E2 10551.102} C_VEL
LIN {X 0,Y 545.62,Z 809.06,A -85,B 0,C 180,E1 10556.309,E2 10556.309} C_VEL
LIN {X 0,Y 545.503,Z 809.06,A -85,B 0,C 180,E1 10561.763,E2 10561.763} C_VEL
LIN {X 0,Y 545.439,Z 809.06,A -85,B 0,C 180,E1 10567.559,E2 10567.559} C_VEL
LIN {X 0,Y 545.418,Z 809.06,A -85,B 0,C 180,E1 10573.923,E2 10573.923} C_VEL
LIN {X 0,Y 545.375,Z 809.06,A -85,B 0,C 180,E1 10580.415,E2 10580.415} C_VEL
LIN {X 0,Y 545.406,Z 809.06,A -85,B 0,C 180,E1 10586.353,E2 10586.353} C_VEL
LIN {X 0,Y 545.698,Z 809.06,A -85,B 0,C 180,E1 10592.399,E2 10592.399} C_VEL
LIN {X 0,Y 545.75,Z 809.06,A -85,B 0,C 180,E1 10597.195,E2 10597.195} C_VEL
LIN {X 0,Y 545.914,Z 809.06,A -85,B 0,C 180,E1 10602.275,E2 10602.275} C_VEL
LIN {X 0,Y 546.02,Z 809.06,A -85,B 0,C 180,E1 10607.21,E2 10607.21} C_VEL
LIN {X 0,Y 546.245,Z 809.06,A -85,B 0,C 180,E1 10613.112,E2 10613.112} C_VEL
LIN {X 0,Y 546.425,Z 809.06,A -85,B 0,C 180,E1 10618.416,E2 10618.416} C_VEL
LIN {X 0,Y 546.374,Z 809.06,A -85,B 0,C 180,E1 10623.171,E2 10623.171} C_VEL
LIN {X 0,Y 546.233,Z 809.06,A -85,B 0,C 180,E1 10627.951,E2 10627.951} C_VEL
LIN {X 0,Y 546.037,Z 809.06,A -85,B 0,C 180,E1 10632.79,E2 10632.79} C_VEL
LIN {X 0,Y 545.905,Z 809.06,A -85,B 0,C 180,E1 10637.727,E2 10637.727} C_VEL
LIN {X 0,Y 545.676,Z 809.06,A -85,B 0,C 180,E1 10642.81,E2 10642.81} C_VEL
LIN {X 0,Y 545.6,Z 809.06,A -85,B 0,C 180,E1 10648.087,E2 10648.087} C_VEL
LIN {X 0,Y 545.486,Z 809.06,A -85,B 0,C 180,E1 10653.784,E2 10653.784} C_VEL
LIN {X 0,Y 545.551,Z 809.06,A -85,B 0,C 180,E1 10654.983,E2 10654.983} C_VEL
LIN {X 0,Y 547.839,Z 814.648,A -85,B 0,C 180,E1 10655.395,E2 10655.395} C_VEL
LIN {X 0,Y 576.794,Z 860.385,A -85,B 0,C 180,E1 10659.623,E2 10659.623} C_VEL
LIN {X 0,Y 597.974,Z 897.517,A -85,B 0,C 180,E1 10662.402,E2 10662.402} C_VEL
LIN {X 0,Y 594.517,Z 948.683,A -85,B 0,C 180,E1 10663.483,E2 10663.483} C_VEL
LIN {X 0,Y 589.63,Z 993.214,A -85,B 0,C 180,E1 10664.928,E2 10664.928} C_VEL
LIN {X 0,Y 583.151,Z 1043.491,A -85,B 0,C 180,E1 10667.222,E2 10667.222} C_VEL
LIN {X 0,Y 576.055,Z 1089.821,A -85,B 0,C 180,E1 10670.07,E2 10670.07} C_VEL
LIN {X 0,Y 572.077,Z 1114.879,A -85,B 0,C 180,E1 10671.934,E2 10671.934} C_VEL
LIN {X 0,Y 566.168,Z 1128.627,A -85,B 0,C 180,E1 10672.888,E2 10672.888} C_VEL
LIN {X 0,Y 560.379,Z 1141.699,A -85,B 0,C 180,E1 10673.897,E2 10673.897} C_VEL
LIN {X 0,Y 554.203,Z 1173.761,A -85,B 0,C 180,E1 10677.461,E2 10677.461} C_VEL
LIN {X 0,Y 548.016,Z 1206.093,A -85,B 0,C 180,E1 10682.04,E2 10682.04} C_VEL
LIN {X 0,Y 543.717,Z 1232.442,A -85,B 0,C 180,E1 10686.764,E2 10686.764} C_VEL
LIN {X 0,Y 540.822,Z 1254.974,A -85,B 0,C 180,E1 10692.094,E2 10692.094} C_VEL
LIN {X 0,Y 539.317,Z 1270.402,A -85,B 0,C 180,E1 10697.041,E2 10697.041} C_VEL
LIN {X 0,Y 538.735,Z 1280.531,A -85,B 0,C 180,E1 10701.932,E2 10701.932} C_VEL
LIN {X 0,Y 538.64,Z 1285.87,A -85,B 0,C 180,E1 10706.777,E2 10706.777} C_VEL
LIN {X 0,Y 538.82,Z 1286.668,A -85,B 0,C 180,E1 10711.6,E2 10711.6} C_VEL
LIN {X 0,Y 538.719,Z 1282.919,A -85,B 0,C 180,E1 10716.435,E2 10716.435} C_VEL
LIN {X 0,Y 539.147,Z 1274.299,A -85,B 0,C 180,E1 10721.307,E2 10721.307} C_VEL
LIN {X 0,Y 540.079,Z 1260.729,A -85,B 0,C 180,E1 10726.24,E2 10726.24} C_VEL
LIN {X 0,Y 542.328,Z 1241.771,A -85,B 0,C 180,E1 10731.229,E2 10731.229} C_VEL
LIN {X 0,Y 545.896,Z 1218.042,A -85,B 0,C 180,E1 10735.954,E2 10735.954} C_VEL
LIN {X 0,Y 551.365,Z 1188.158,A -85,B 0,C 180,E1 10740.643,E2 10740.643} C_VEL
LIN {X 0,Y 558.06,Z 1154.109,A -85,B 0,C 180,E1 10744.828,E2 10744.828} C_VEL
LIN {X 0,Y 562.675,Z 1127.464,A -85,B 0,C 180,E1 10747.336,E2 10747.336} C_VEL
LIN {X 0,Y 569.251,Z 1082.7,A -85,B 0,C 180,E1 10750.58,E2 10750.58} C_VEL
LIN {X 0,Y 575.325,Z 1036.146,A -85,B 0,C 180,E1 10753.217,E2 10753.217} C_VEL
LIN {X 0,Y 581.207,Z 982.411,A -85,B 0,C 180,E1 10755.462,E2 10755.462} C_VEL
LIN {X 0,Y 585.712,Z 931.767,A -85,B 0,C 180,E1 10756.924,E2 10756.924} C_VEL
LIN {X 0,Y 587.524,Z 899.326,A -85,B 0,C 180,E1 10757.6,E2 10757.6} C_VEL
LIN {X 0,Y 570.32,Z 870.38,A -85,B 0,C 180,E1 10759.526,E2 10759.526} C_VEL
LIN {X 0,Y 552.909,Z 835.945,A -85,B 0,C 180,E1 10761.87,E2 10761.87} C_VEL
LIN {X 0,Y 540.503,Z 815.283,A -85,B 0,C 180,E1 10763.928,E2 10763.928} C_VEL
LIN {X 0,Y 537.532,Z 809.758,A -85,B 0,C 180,E1 10764.564,E2 10764.564} C_VEL
LIN {X 0,Y 537.507,Z 809.06,A -85,B 0,C 180,E1 10770.617,E2 10770.617} C_VEL
LIN {X 0,Y 537.638,Z 809.471,A -85,B 0,C 180,E1 10772.129,E2 10772.129} C_VEL
LIN {X 0,Y 540.382,Z 815.03,A -85,B 0,C 180,E1 10772.834,E2 10772.834} C_VEL
LIN {X 0,Y 551.882,Z 835.6,A -85,B 0,C 180,E1 10775.28,E2 10775.28} C_VEL
LIN {X 0,Y 569.095,Z 875.308,A -85,B 0,C 180,E1 10779.235,E2 10779.235} C_VEL
LIN {X 0,Y 578.139,Z 900.257,A -85,B 0,C 180,E1 10781.722,E2 10781.722} C_VEL
LIN {X 0,Y 571.348,Z 940.622,A -85,B 0,C 180,E1 10784.271,E2 10784.271} C_VEL
LIN {X 0,Y 563.666,Z 978.44,A -85,B 0,C 180,E1 10787.419,E2 10787.419} C_VEL
LIN {X 0,Y 555.228,Z 1018.565,A -85,B 0,C 180,E1 10791.785,E2 10791.785} C_VEL
LIN {X 0,Y 549.102,Z 1050.11,A -85,B 0,C 180,E1 10796.055,E2 10796.055} C_VEL
LIN {X 0,Y 544.354,Z 1078.164,A -85,B 0,C 180,E1 10800.879,E2 10800.879} C_VEL
LIN {X 0,Y 541.274,Z 1099.572,A -85,B 0,C 180,E1 10805.606,E2 10805.606} C_VEL
LIN {X 0,Y 539.667,Z 1116.206,A -85,B 0,C 180,E1 10810.485,E2 10810.485} C_VEL
LIN {X 0,Y 538.789,Z 1128.043,A -85,B 0,C 180,E1 10815.451,E2 10815.451} C_VEL
LIN {X 0,Y 538.362,Z 1134.256,A -85,B 0,C 180,E1 10819.681,E2 10819.681} C_VEL
LIN {X 0,Y 537.943,Z 1136.998,A -85,B 0,C 180,E1 10824.918,E2 10824.918} C_VEL
LIN {X 0,Y 538.375,Z 1134.128,A -85,B 0,C 180,E1 10830.343,E2 10830.343} C_VEL
LIN {X 0,Y 538.945,Z 1126.837,A -85,B 0,C 180,E1 10835.097,E2 10835.097} C_VEL
LIN {X 0,Y 539.821,Z 1114.307,A -85,B 0,C 180,E1 10840.074,E2 10840.074} C_VEL
LIN {X 0,Y 541.736,Z 1096.311,A -85,B 0,C 180,E1 10845.112,E2 10845.112} C_VEL
LIN {X 0,Y 545.259,Z 1072.453,A -85,B 0,C 180,E1 10850.123,E2 10850.123} C_VEL
LIN {X 0,Y 550.493,Z 1042.696,A -85,B 0,C 180,E1 10854.957,E2 10854.957} C_VEL
LIN {X 0,Y 557.269,Z 1007.776,A -85,B 0,C 180,E1 10859.388,E2 10859.388} C_VEL
LIN {X 0,Y 564.882,Z 971.685,A -85,B 0,C 180,E1 10863.057,E2 10863.057} C_VEL
LIN {X 0,Y 572.409,Z 933.348,A -85,B 0,C 180,E1 10866.104,E2 10866.104} C_VEL
LIN {X 0,Y 578.129,Z 900.316,A -85,B 0,C 180,E1 10868.187,E2 10868.187} C_VEL
LIN {X 0,Y 565.547,Z 865.889,A -85,B 0,C 180,E1 10871.71,E2 10871.71} C_VEL
LIN {X 0,Y 548.851,Z 830.597,A -85,B 0,C 180,E1 10875.489,E2 10875.489} C_VEL
LIN {X 0,Y 538.078,Z 809.76,A -85,B 0,C 180,E1 10877.745,E2 10877.745} C_VEL
LIN {X 0,Y 538.319,Z 809.06,A -85,B 0,C 180,E1 10881.939,E2 10881.939} C_VEL
LIN {X 0,Y 538.52,Z 809.06,A -85,B 0,C 180,E1 10886.79,E2 10886.79} C_VEL
LIN {X 0,Y 538.533,Z 809.06,A -85,B 0,C 180,E1 10891.614,E2 10891.614} C_VEL
LIN {X 0,Y 538.393,Z 809.06,A -85,B 0,C 180,E1 10896.452,E2 10896.452} C_VEL
LIN {X 0,Y 538.178,Z 809.06,A -85,B 0,C 180,E1 10901.341,E2 10901.341} C_VEL
LIN {X 0,Y 537.993,Z 809.06,A -85,B 0,C 180,E1 10907.273,E2 10907.273} C_VEL
LIN {X 0,Y 537.774,Z 809.06,A -85,B 0,C 180,E1 10913.172,E2 10913.172} C_VEL
LIN {X 0,Y 537.617,Z 809.06,A -85,B 0,C 180,E1 10919.395,E2 10919.395} C_VEL
LIN {X 0,Y 537.528,Z 809.06,A -85,B 0,C 180,E1 10925.395,E2 10925.395} C_VEL
LIN {X 0,Y 537.43,Z 809.06,A -85,B 0,C 180,E1 10930.615,E2 10930.615} C_VEL
LIN {X 0,Y 537.431,Z 809.06,A -85,B 0,C 180,E1 10935.343,E2 10935.343} C_VEL
LIN {X 0,Y 537.443,Z 809.06,A -85,B 0,C 180,E1 10941.938,E2 10941.938} C_VEL
LIN {X 0,Y 537.496,Z 809.06,A -85,B 0,C 180,E1 10947.716,E2 10947.716} C_VEL
LIN {X 0,Y 537.76,Z 809.06,A -85,B 0,C 180,E1 10953.285,E2 10953.285} C_VEL
LIN {X 0,Y 537.87,Z 809.06,A -85,B 0,C 180,E1 10958.581,E2 10958.581} C_VEL
LIN {X 0,Y 537.989,Z 809.06,A -85,B 0,C 180,E1 10963.689,E2 10963.689} C_VEL
LIN {X 0,Y 538.178,Z 809.06,A -85,B 0,C 180,E1 10969.361,E2 10969.361} C_VEL
LIN {X 0,Y 538.457,Z 809.06,A -85,B 0,C 180,E1 10975.171,E2 10975.171} C_VEL
LIN {X 0,Y 538.737,Z 809.06,A -85,B 0,C 180,E1 10980.001,E2 10980.001} C_VEL
LIN {X 0,Y 538.393,Z 809.06,A -85,B 0,C 180,E1 10986.446,E2 10986.446} C_VEL
LIN {X 0,Y 538.186,Z 809.06,A -85,B 0,C 180,E1 10991.335,E2 10991.335} C_VEL
LIN {X 0,Y 537.969,Z 809.06,A -85,B 0,C 180,E1 10997.234,E2 10997.234} C_VEL
LIN {X 0,Y 537.745,Z 809.06,A -85,B 0,C 180,E1 11003.166,E2 11003.166} C_VEL
LIN {X 0,Y 537.586,Z 809.06,A -85,B 0,C 180,E1 11009.371,E2 11009.371} C_VEL
LIN {X 0,Y 537.591,Z 809.464,A -85,B 0,C 180,E1 11013.98,E2 11013.98} C_VEL
LIN {X 0,Y 540.24,Z 814.955,A -85,B 0,C 180,E1 11014.455,E2 11014.455} C_VEL
LIN {X 0,Y 569.49,Z 860.962,A -85,B 0,C 180,E1 11018.854,E2 11018.854} C_VEL
LIN {X 0,Y 592.028,Z 900.542,A -85,B 0,C 180,E1 11021.907,E2 11021.907} C_VEL
LIN {X 0,Y 588.411,Z 950.604,A -85,B 0,C 180,E1 11023.023,E2 11023.023} C_VEL
LIN {X 0,Y 582.969,Z 997.227,A -85,B 0,C 180,E1 11024.588,E2 11024.588} C_VEL
LIN {X 0,Y 576.432,Z 1045.088,A -85,B 0,C 180,E1 11026.842,E2 11026.842} C_VEL
LIN {X 0,Y 568.773,Z 1092.904,A -85,B 0,C 180,E1 11029.856,E2 11029.856} C_VEL
LIN {X 0,Y 561.927,Z 1133.224,A -85,B 0,C 180,E1 11033.115,E2 11033.115} C_VEL
LIN {X 0,Y 560.379,Z 1141.699,A -85,B 0,C 180,E1 11033.897,E2 11033.897} C_VEL
LIN {X 0,Y 554.528,Z 1154.516,A -85,B 0,C 180,E1 11034.974,E2 11034.974} C_VEL
LIN {X 0,Y 548.594,Z 1166.673,A -85,B 0,C 180,E1 11036.136,E2 11036.136} C_VEL
LIN {X 0,Y 541.983,Z 1199.439,A -85,B 0,C 180,E1 11040.561,E2 11040.561} C_VEL
LIN {X 0,Y 536.78,Z 1228.129,A -85,B 0,C 180,E1 11045.563,E2 11045.563} C_VEL
LIN {X 0,Y 533.501,Z 1250.368,A -85,B 0,C 180,E1 11050.554,E2 11050.554} C_VEL
LIN {X 0,Y 531.781,Z 1266.968,A -85,B 0,C 180,E1 11055.597,E2 11055.597} C_VEL
LIN {X 0,Y 530.97,Z 1277.653,A -85,B 0,C 180,E1 11060.162,E2 11060.162} C_VEL
LIN {X 0,Y 530.709,Z 1284.764,A -85,B 0,C 180,E1 11065.205,E2 11065.205} C_VEL
LIN {X 0,Y 530.791,Z 1287,A -85,B 0,C 180,E1 11069.993,E2 11069.993} C_VEL
LIN {X 0,Y 530.701,Z 1284.662,A -85,B 0,C 180,E1 11074.893,E2 11074.893} C_VEL
LIN {X 0,Y 530.959,Z 1277.679,A -85,B 0,C 180,E1 11079.825,E2 11079.825} C_VEL
LIN {X 0,Y 531.994,Z 1265.183,A -85,B 0,C 180,E1 11085.052,E2 11085.052} C_VEL
LIN {X 0,Y 533.883,Z 1247.466,A -85,B 0,C 180,E1 11090.16,E2 11090.16} C_VEL
LIN {X 0,Y 537.372,Z 1224.136,A -85,B 0,C 180,E1 11095.225,E2 11095.225} C_VEL
LIN {X 0,Y 542.564,Z 1196.623,A -85,B 0,C 180,E1 11099.848,E2 11099.848} C_VEL
LIN {X 0,Y 549.075,Z 1164.444,A -85,B 0,C 180,E1 11104.121,E2 11104.121} C_VEL
LIN {X 0,Y 555.135,Z 1128.157,A -85,B 0,C 180,E1 11107.566,E2 11107.566} C_VEL
LIN {X 0,Y 561.693,Z 1084.81,A -85,B 0,C 180,E1 11110.783,E2 11110.783} C_VEL
LIN {X 0,Y 568.138,Z 1037.844,A -85,B 0,C 180,E1 11113.511,E2 11113.511} C_VEL
LIN {X 0,Y 573.925,Z 986.975,A -85,B 0,C 180,E1 11115.715,E2 11115.715} C_VEL
LIN {X 0,Y 579.083,Z 934.312,A -85,B 0,C 180,E1 11117.319,E2 11117.319} C_VEL
LIN {X 0,Y 580.959,Z 902.362,A -85,B 0,C 180,E1 11118.017,E2 11118.017} C_VEL
LIN {X 0,Y 565.111,Z 875.071,A -85,B 0,C 180,E1 11119.892,E2 11119.892} C_VEL
LIN {X 0,Y 548.461,Z 841.344,A -85,B 0,C 180,E1 11122.256,E2 11122.256} C_VEL
LIN {X 0,Y 537.055,Z 821.769,A -85,B 0,C 180,E1 11124.263,E2 11124.263} C_VEL
LIN {X 0,Y 532.504,Z 815.232,A -85,B 0,C 180,E1 11125.282,E2 11125.282} C_VEL
LIN {X 0,Y 529.53,Z 809.623,A -85,B 0,C 180,E1 11126.213,E2 11126.213} C_VEL
LIN {X 0,Y 529.623,Z 809.703,A -85,B 0,C 180,E1 11130.456,E2 11130.456} C_VEL
LIN {X 0,Y 532.563,Z 815.151,A -85,B 0,C 180,E1 11131.421,E2 11131.421} C_VEL
LIN {X 0,Y 534.602,Z 818.154,A -85,B 0,C 180,E1 11131.986,E2 11131.986} C_VEL
LIN {X 0,Y 544.109,Z 834.907,A -85,B 0,C 180,E1 11134.243,E2 11134.243} C_VEL
LIN {X 0,Y 558.386,Z 866.958,A -85,B 0,C 180,E1 11137.621,E2 11137.621} C_VEL
LIN {X 0,Y 571.683,Z 903.118,A -85,B 0,C 180,E1 11141.303,E2 11141.303} C_VEL
LIN {X 0,Y 564.902,Z 943.159,A -85,B 0,C 180,E1 11143.888,E2 11143.888} C_VEL
LIN {X 0,Y 556.993,Z 980.9,A -85,B 0,C 180,E1 11147.067,E2 11147.067} C_VEL
LIN {X 0,Y 549.519,Z 1014.053,A -85,B 0,C 180,E1 11150.703,E2 11150.703} C_VEL
LIN {X 0,Y 541.669,Z 1051.189,A -85,B 0,C 180,E1 11155.8,E2 11155.8} C_VEL
LIN {X 0,Y 536.711,Z 1078.919,A -85,B 0,C 180,E1 11160.668,E2 11160.668} C_VEL
LIN {X 0,Y 533.413,Z 1101.029,A -85,B 0,C 180,E1 11165.689,E2 11165.689} C_VEL
LIN {X 0,Y 531.764,Z 1117.206,A -85,B 0,C 180,E1 11170.619,E2 11170.619} C_VEL
LIN {X 0,Y 530.857,Z 1128.736,A -85,B 0,C 180,E1 11175.687,E2 11175.687} C_VEL
LIN {X 0,Y 530.399,Z 1134.631,A -85,B 0,C 180,E1 11179.989,E2 11179.989} C_VEL
LIN {X 0,Y 530.033,Z 1136.944,A -85,B 0,C 180,E1 11185.315,E2 11185.315} C_VEL
LIN {X 0,Y 530.254,Z 1135.417,A -85,B 0,C 180,E1 11188.974,E2 11188.974} C_VEL
LIN {X 0,Y 530.853,Z 1130.38,A -85,B 0,C 180,E1 11193.247,E2 11193.247} C_VEL
LIN {X 0,Y 531.512,Z 1120.786,A -85,B 0,C 180,E1 11197.933,E2 11197.933} C_VEL
LIN {X 0,Y 533.055,Z 1104.727,A -85,B 0,C 180,E1 11203.209,E2 11203.209} C_VEL
LIN {X 0,Y 535.887,Z 1084.154,A -85,B 0,C 180,E1 11208.165,E2 11208.165} C_VEL
LIN {X 0,Y 540.337,Z 1057.929,A -85,B 0,C 180,E1 11213.036,E2 11213.036} C_VEL
LIN {X 0,Y 546.516,Z 1026.711,A -85,B 0,C 180,E1 11217.579,E2 11217.579} C_VEL
LIN {X 0,Y 554.32,Z 991.412,A -85,B 0,C 180,E1 11221.72,E2 11221.72} C_VEL
LIN {X 0,Y 562.626,Z 952.454,A -85,B 0,C 180,E1 11225.247,E2 11225.247} C_VEL
LIN {X 0,Y 570.36,Z 910.798,A -85,B 0,C 180,E1 11228.137,E2 11228.137} C_VEL
LIN {X 0,Y 571.442,Z 902.33,A -85,B 0,C 180,E1 11228.686,E2 11228.686} C_VEL
LIN {X 0,Y 558.605,Z 867.104,A -85,B 0,C 180,E1 11232.378,E2 11232.378} C_VEL
LIN {X 0,Y 541.719,Z 831.666,A -85,B 0,C 180,E1 11236.292,E2 11236.292} C_VEL
LIN {X 0,Y 530.283,Z 809.756,A -85,B 0,C 180,E1 11238.746,E2 11238.746} C_VEL
LIN {X 0,Y 530.479,Z 809.06,A -85,B 0,C 180,E1 11243.464,E2 11243.464} C_VEL
LIN {X 0,Y 530.568,Z 809.06,A -85,B 0,C 180,E1 11248.375,E2 11248.375} C_VEL
LIN {X 0,Y 530.502,Z 809.06,A -85,B 0,C 180,E1 11253.272,E2 11253.272} C_VEL
LIN {X 0,Y 530.384,Z 809.06,A -85,B 0,C 180,E1 11258.196,E2 11258.196} C_VEL
LIN {X 0,Y 530.178,Z 809.06,A -85,B 0,C 180,E1 11264.309,E2 11264.309} C_VEL
LIN {X 0,Y 529.997,Z 809.06,A -85,B 0,C 180,E1 11270.013,E2 11270.013} C_VEL
LIN {X 0,Y 529.78,Z 809.06,A -85,B 0,C 180,E1 11275.337,E2 11275.337} C_VEL
LIN {X 0,Y 529.627,Z 809.06,A -85,B 0,C 180,E1 11281.144,E2 11281.144} C_VEL
LIN {X 0,Y 529.54,Z 809.06,A -85,B 0,C 180,E1 11286.971,E2 11286.971} C_VEL
LIN {X 0,Y 529.535,Z 809.06,A -85,B 0,C 180,E1 11293.233,E2 11293.233} C_VEL
LIN {X 0,Y 529.457,Z 809.06,A -85,B 0,C 180,E1 11298.976,E2 11298.976} C_VEL
LIN {X 0,Y 529.522,Z 809.06,A -85,B 0,C 180,E1 11305.202,E2 11305.202} C_VEL
LIN {X 0,Y 529.749,Z 809.06,A -85,B 0,C 180,E1 11310.996,E2 11310.996} C_VEL
LIN {X 0,Y 529.867,Z 809.06,A -85,B 0,C 180,E1 11316.471,E2 11316.471} C_VEL
LIN {X 0,Y 530.045,Z 809.06,A -85,B 0,C 180,E1 11321.726,E2 11321.726} C_VEL
LIN {X 0,Y 530.174,Z 809.06,A -85,B 0,C 180,E1 11326.821,E2 11326.821} C_VEL
LIN {X 0,Y 530.434,Z 809.06,A -85,B 0,C 180,E1 11331.812,E2 11331.812} C_VEL
LIN {X 0,Y 530.621,Z 809.06,A -85,B 0,C 180,E1 11336.736,E2 11336.736} C_VEL
LIN {X 0,Y 530.756,Z 809.06,A -85,B 0,C 180,E1 11341.632,E2 11341.632} C_VEL
LIN {X 0,Y 530.492,Z 809.06,A -85,B 0,C 180,E1 11346.543,E2 11346.543} C_VEL
LIN {X 0,Y 530.259,Z 809.06,A -85,B 0,C 180,E1 11351.506,E2 11351.506} C_VEL
LIN {X 0,Y 530.096,Z 809.06,A -85,B 0,C 180,E1 11356.562,E2 11356.562} C_VEL
LIN {X 0,Y 529.894,Z 809.06,A -85,B 0,C 180,E1 11361.759,E2 11361.759} C_VEL
LIN {X 0,Y 529.702,Z 809.06,A -85,B 0,C 180,E1 11367.818,E2 11367.818} C_VEL
LIN {X 0,Y 529.666,Z 809.839,A -85,B 0,C 180,E1 11372.929,E2 11372.929} C_VEL
LIN {X 0,Y 532.579,Z 815.199,A -85,B 0,C 180,E1 11373.441,E2 11373.441} C_VEL
LIN {X 0,Y 559.712,Z 857.712,A -85,B 0,C 180,E1 11377.708,E2 11377.708} C_VEL
LIN {X 0,Y 586.308,Z 903.907,A -85,B 0,C 180,E1 11381.426,E2 11381.426} C_VEL
LIN {X 0,Y 582,Z 955.228,A -85,B 0,C 180,E1 11382.629,E2 11382.629} C_VEL
LIN {X 0,Y 576.012,Z 1003.687,A -85,B 0,C 180,E1 11384.335,E2 11384.335} C_VEL
LIN {X 0,Y 568.661,Z 1053.083,A -85,B 0,C 180,E1 11386.821,E2 11386.821} C_VEL
LIN {X 0,Y 561.226,Z 1097.287,A -85,B 0,C 180,E1 11389.738,E2 11389.738} C_VEL
LIN {X 0,Y 553.208,Z 1141.686,A -85,B 0,C 180,E1 11393.522,E2 11393.522} C_VEL
LIN {X 0,Y 548.594,Z 1166.673,A -85,B 0,C 180,E1 11396.136,E2 11396.136} C_VEL
LIN {X 0,Y 542.81,Z 1178.434,A -85,B 0,C 180,E1 11397.36,E2 11397.36} C_VEL
LIN {X 0,Y 536.89,Z 1189.53,A -85,B 0,C 180,E1 11398.661,E2 11398.661} C_VEL
LIN {X 0,Y 530.701,Z 1220.365,A -85,B 0,C 180,E1 11403.686,E2 11403.686} C_VEL
LIN {X 0,Y 526.688,Z 1244.181,A -85,B 0,C 180,E1 11408.718,E2 11408.718} C_VEL
LIN {X 0,Y 524.396,Z 1262.014,A -85,B 0,C 180,E1 11413.676,E2 11413.676} C_VEL
LIN {X 0,Y 523.314,Z 1274.268,A -85,B 0,C 180,E1 11418.332,E2 11418.332} C_VEL
LIN {X 0,Y 522.946,Z 1282.902,A -85,B 0,C 180,E1 11423.356,E2 11423.356} C_VEL
LIN {X 0,Y 522.766,Z 1286.664,A -85,B 0,C 180,E1 11428.337,E2 11428.337} C_VEL
LIN {X 0,Y 523.013,Z 1286.668,A -85,B 0,C 180,E1 11431.649,E2 11431.649} C_VEL
LIN {X 0,Y 522.93,Z 1282.919,A -85,B 0,C 180,E1 11436.63,E2 11436.63} C_VEL
LIN {X 0,Y 523.392,Z 1274.299,A -85,B 0,C 180,E1 11441.652,E2 11441.652} C_VEL
LIN {X 0,Y 524.495,Z 1260.727,A -85,B 0,C 180,E1 11446.737,E2 11446.737} C_VEL
LIN {X 0,Y 527.06,Z 1241.772,A -85,B 0,C 180,E1 11451.875,E2 11451.875} C_VEL
LIN {X 0,Y 531.271,Z 1217.306,A -85,B 0,C 180,E1 11456.864,E2 11456.864} C_VEL
LIN {X 0,Y 537.274,Z 1187.892,A -85,B 0,C 180,E1 11461.581,E2 11461.581} C_VEL
LIN {X 0,Y 541.546,Z 1164.463,A -85,B 0,C 180,E1 11464.385,E2 11464.385} C_VEL
LIN {X 0,Y 548.128,Z 1125.611,A -85,B 0,C 180,E1 11468.069,E2 11468.069} C_VEL
LIN {X 0,Y 554.978,Z 1081.796,A -85,B 0,C 180,E1 11471.327,E2 11471.327} C_VEL
LIN {X 0,Y 561.612,Z 1034.736,A -85,B 0,C 180,E1 11474.055,E2 11474.055} C_VEL
LIN {X 0,Y 567.727,Z 983.046,A -85,B 0,C 180,E1 11476.281,E2 11476.281} C_VEL
LIN {X 0,Y 572.929,Z 931.468,A -85,B 0,C 180,E1 11477.846,E2 11477.846} C_VEL
LIN {X 0,Y 574.449,Z 905.528,A -85,B 0,C 180,E1 11478.441,E2 11478.441} C_VEL
LIN {X 0,Y 559.662,Z 879.121,A -85,B 0,C 180,E1 11480.306,E2 11480.306} C_VEL
LIN {X 0,Y 543.562,Z 845.833,A -85,B 0,C 180,E1 11482.736,E2 11482.736} C_VEL
LIN {X 0,Y 533.338,Z 827.834,A -85,B 0,C 180,E1 11484.68,E2 11484.68} C_VEL
LIN {X 0,Y 529.272,Z 821.724,A -85,B 0,C 180,E1 11485.695,E2 11485.695} C_VEL
LIN {X 0,Y 526.262,Z 816.257,A -85,B 0,C 180,E1 11486.826,E2 11486.826} C_VEL
LIN {X 0,Y 524.51,Z 815.216,A -85,B 0,C 180,E1 11488.086,E2 11488.086} C_VEL
LIN {X 0,Y 526.889,Z 816.472,A -85,B 0,C 180,E1 11490.066,E2 11490.066} C_VEL
LIN {X 0,Y 530.135,Z 822.606,A -85,B 0,C 180,E1 11491.312,E2 11491.312} C_VEL
LIN {X 0,Y 539.504,Z 839.999,A -85,B 0,C 180,E1 11493.824,E2 11493.824} C_VEL
LIN {X 0,Y 553.373,Z 872.907,A -85,B 0,C 180,E1 11497.407,E2 11497.407} C_VEL
LIN {X 0,Y 565.253,Z 905.975,A -85,B 0,C 180,E1 11500.868,E2 11500.868} C_VEL
LIN {X 0,Y 558.463,Z 945.726,A -85,B 0,C 180,E1 11503.495,E2 11503.495} C_VEL
LIN {X 0,Y 550.332,Z 983.354,A -85,B 0,C 180,E1 11506.706,E2 11506.706} C_VEL
LIN {X 0,Y 542.62,Z 1016.408,A -85,B 0,C 180,E1 11510.381,E2 11510.381} C_VEL
LIN {X 0,Y 533.471,Z 1056.098,A -85,B 0,C 180,E1 11516.142,E2 11516.142} C_VEL
LIN {X 0,Y 528.61,Z 1082.278,A -85,B 0,C 180,E1 11520.983,E2 11520.983} C_VEL
LIN {X 0,Y 525.296,Z 1103.949,A -85,B 0,C 180,E1 11526.192,E2 11526.192} C_VEL
LIN {X 0,Y 523.711,Z 1119.421,A -85,B 0,C 180,E1 11531.225,E2 11531.225} C_VEL
LIN {X 0,Y 522.942,Z 1129.426,A -85,B 0,C 180,E1 11535.931,E2 11535.931} C_VEL
LIN {X 0,Y 522.418,Z 1134.951,A -85,B 0,C 180,E1 11540.308,E2 11540.308} C_VEL
LIN {X 0,Y 522.097,Z 1136.877,A -85,B 0,C 180,E1 11545.728,E2 11545.728} C_VEL
LIN {X 0,Y 522.685,Z 1133.143,A -85,B 0,C 180,E1 11551.355,E2 11551.355} C_VEL
LIN {X 0,Y 523.285,Z 1125.507,A -85,B 0,C 180,E1 11556.059,E2 11556.059} C_VEL
LIN {X 0,Y 524.345,Z 1112.75,A -85,B 0,C 180,E1 11561.065,E2 11561.065} C_VEL
LIN {X 0,Y 526.943,Z 1093.029,A -85,B 0,C 180,E1 11566.52,E2 11566.52} C_VEL
LIN {X 0,Y 531.302,Z 1067.704,A -85,B 0,C 180,E1 11571.75,E2 11571.75} C_VEL
LIN {X 0,Y 537.31,Z 1037.488,A -85,B 0,C 180,E1 11576.593,E2 11576.593} C_VEL
LIN {X 0,Y 544.827,Z 1004.913,A -85,B 0,C 180,E1 11580.82,E2 11580.82} C_VEL
LIN {X 0,Y 553.352,Z 967.375,A -85,B 0,C 180,E1 11584.572,E2 11584.572} C_VEL
LIN {X 0,Y 561.954,Z 924.974,A -85,B 0,C 180,E1 11587.809,E2 11587.809} C_VEL
LIN {X 0,Y 565.076,Z 905.61,A -85,B 0,C 180,E1 11589.062,E2 11589.062} C_VEL
LIN {X 0,Y 552.315,Z 869.909,A -85,B 0,C 180,E1 11592.903,E2 11592.903} C_VEL
LIN {X 0,Y 534.628,Z 832.523,A -85,B 0,C 180,E1 11597.135,E2 11597.135} C_VEL
LIN {X 0,Y 522.459,Z 809.991,A -85,B 0,C 180,E1 11599.791,E2 11599.791} C_VEL
LIN {X 0,Y 522.411,Z 809.06,A -85,B 0,C 180,E1 11600.013,E2 11600.013} C_VEL
LIN {X 0,Y 522.643,Z 809.06,A -85,B 0,C 180,E1 11605.031,E2 11605.031} C_VEL
LIN {X 0,Y 522.851,Z 809.06,A -85,B 0,C 180,E1 11610.007,E2 11610.007} C_VEL
LIN {X 0,Y 522.562,Z 809.06,A -85,B 0,C 180,E1 11616.649,E2 11616.649} C_VEL
LIN {X 0,Y 522.341,Z 809.06,A -85,B 0,C 180,E1 11621.69,E2 11621.69} C_VEL
LIN {X 0,Y 522.153,Z 809.06,A -85,B 0,C 180,E1 11627.267,E2 11627.267} C_VEL
LIN {X 0,Y 521.947,Z 809.06,A -85,B 0,C 180,E1 11632.126,E2 11632.126} C_VEL
LIN {X 0,Y 521.851,Z 809.06,A -85,B 0,C 180,E1 11637.607,E2 11637.607} C_VEL
LIN {X 0,Y 521.705,Z 809.06,A -85,B 0,C 180,E1 11643.396,E2 11643.396} C_VEL
LIN {X 0,Y 521.62,Z 809.06,A -85,B 0,C 180,E1 11649.6,E2 11649.6} C_VEL
LIN {X 0,Y 521.6,Z 809.06,A -85,B 0,C 180,E1 11655.955,E2 11655.955} C_VEL
LIN {X 0,Y 521.549,Z 809.06,A -85,B 0,C 180,E1 11661.478,E2 11661.478} C_VEL
LIN {X 0,Y 521.681,Z 809.06,A -85,B 0,C 180,E1 11667.151,E2 11667.151} C_VEL
LIN {X 0,Y 521.891,Z 809.06,A -85,B 0,C 180,E1 11672.405,E2 11672.405} C_VEL
LIN {X 0,Y 522.014,Z 809.06,A -85,B 0,C 180,E1 11677.897,E2 11677.897} C_VEL
LIN {X 0,Y 522.149,Z 809.06,A -85,B 0,C 180,E1 11683.18,E2 11683.18} C_VEL
LIN {X 0,Y 522.402,Z 809.06,A -85,B 0,C 180,E1 11689.598,E2 11689.598} C_VEL
LIN {X 0,Y 522.633,Z 809.06,A -85,B 0,C 180,E1 11695.025,E2 11695.025} C_VEL
LIN {X 0,Y 522.936,Z 809.06,A -85,B 0,C 180,E1 11700.001,E2 11700.001} C_VEL
LIN {X 0,Y 522.691,Z 809.06,A -85,B 0,C 180,E1 11704.976,E2 11704.976} C_VEL
LIN {X 0,Y 522.401,Z 809.06,A -85,B 0,C 180,E1 11710.401,E2 11710.401} C_VEL
LIN {X 0,Y 522.156,Z 809.06,A -85,B 0,C 180,E1 11716.821,E2 11716.821} C_VEL
LIN {X 0,Y 521.949,Z 809.06,A -85,B 0,C 180,E1 11722.108,E2 11722.108} C_VEL
LIN {X 0,Y 521.83,Z 809.06,A -85,B 0,C 180,E1 11727.6,E2 11727.6} C_VEL
LIN {X 0,Y 521.7,Z 809.402,A -85,B 0,C 180,E1 11731.822,E2 11731.822} C_VEL
LIN {X 0,Y 524.25,Z 814.857,A -85,B 0,C 180,E1 11732.32,E2 11732.32} C_VEL
LIN {X 0,Y 549.356,Z 853.372,A -85,B 0,C 180,E1 11736.413,E2 11736.413} C_VEL
LIN {X 0,Y 572.139,Z 892.409,A -85,B 0,C 180,E1 11739.763,E2 11739.763} C_VEL
LIN {X 0,Y 580.513,Z 908.463,A -85,B 0,C 180,E1 11740.978,E2 11740.978} C_VEL
LIN {X 0,Y 575.306,Z 962.65,A -85,B 0,C 180,E1 11742.308,E2 11742.308} C_VEL
LIN {X 0,Y 568.802,Z 1011.164,A -85,B 0,C 180,E1 11744.162,E2 11744.162} C_VEL
LIN {X 0,Y 561.213,Z 1059.159,A -85,B 0,C 180,E1 11746.687,E2 11746.687} C_VEL
LIN {X 0,Y 552.898,Z 1105.299,A -85,B 0,C 180,E1 11749.926,E2 11749.926} C_VEL
LIN {X 0,Y 545.296,Z 1145.855,A -85,B 0,C 180,E1 11753.553,E2 11753.553} C_VEL
LIN {X 0,Y 538.238,Z 1182.974,A -85,B 0,C 180,E1 11757.756,E2 11757.756} C_VEL
LIN {X 0,Y 536.89,Z 1189.53,A -85,B 0,C 180,E1 11758.661,E2 11758.661} C_VEL
LIN {X 0,Y 531.108,Z 1200.241,A -85,B 0,C 180,E1 11760.034,E2 11760.034} C_VEL
LIN {X 0,Y 525.352,Z 1210.211,A -85,B 0,C 180,E1 11761.453,E2 11761.453} C_VEL
LIN {X 0,Y 520.458,Z 1235.896,A -85,B 0,C 180,E1 11766.464,E2 11766.464} C_VEL
LIN {X 0,Y 517.301,Z 1257.199,A -85,B 0,C 180,E1 11771.893,E2 11771.893} C_VEL
LIN {X 0,Y 515.594,Z 1272.346,A -85,B 0,C 180,E1 11777.296,E2 11777.296} C_VEL
LIN {X 0,Y 515.063,Z 1281.73,A -85,B 0,C 180,E1 11782.407,E2 11782.407} C_VEL
LIN {X 0,Y 514.933,Z 1285.87,A -85,B 0,C 180,E1 11786.629,E2 11786.629} C_VEL
LIN {X 0,Y 515.106,Z 1286.668,A -85,B 0,C 180,E1 11791.674,E2 11791.674} C_VEL
LIN {X 0,Y 515.051,Z 1282.919,A -85,B 0,C 180,E1 11796.732,E2 11796.732} C_VEL
LIN {X 0,Y 515.518,Z 1274.298,A -85,B 0,C 180,E1 11801.833,E2 11801.833} C_VEL
LIN {X 0,Y 516.729,Z 1260.726,A -85,B 0,C 180,E1 11806.996,E2 11806.996} C_VEL
LIN {X 0,Y 519.46,Z 1241.773,A -85,B 0,C 180,E1 11812.212,E2 11812.212} C_VEL
LIN {X 0,Y 524.178,Z 1216.264,A -85,B 0,C 180,E1 11817.459,E2 11817.459} C_VEL
LIN {X 0,Y 528.816,Z 1193.264,A -85,B 0,C 180,E1 11821.184,E2 11821.184} C_VEL
LIN {X 0,Y 535.222,Z 1157.421,A -85,B 0,C 180,E1 11825.37,E2 11825.37} C_VEL
LIN {X 0,Y 542.203,Z 1116.534,A -85,B 0,C 180,E1 11829.112,E2 11829.112} C_VEL
LIN {X 0,Y 549.516,Z 1071.461,A -85,B 0,C 180,E1 11832.353,E2 11832.353} C_VEL
LIN {X 0,Y 556.106,Z 1024.643,A -85,B 0,C 180,E1 11834.939,E2 11834.939} C_VEL
LIN {X 0,Y 562.153,Z 974.821,A -85,B 0,C 180,E1 11837.014,E2 11837.014} C_VEL
LIN {X 0,Y 567.187,Z 924.52,A -85,B 0,C 180,E1 11838.48,E2 11838.48} C_VEL
LIN {X 0,Y 567.966,Z 908.625,A -85,B 0,C 180,E1 11838.881,E2 11838.881} C_VEL
LIN {X 0,Y 554.385,Z 883.639,A -85,B 0,C 180,E1 11840.69,E2 11840.69} C_VEL
LIN {X 0,Y 539.249,Z 851.196,A -85,B 0,C 180,E1 11843.143,E2 11843.143} C_VEL
LIN {X 0,Y 529.827,Z 833.923,A -85,B 0,C 180,E1 11845.099,E2 11845.099} C_VEL
LIN {X 0,Y 524.589,Z 823.944,A -85,B 0,C 180,E1 11846.894,E2 11846.894} C_VEL
LIN {X 0,Y 522.914,Z 822.962,A -85,B 0,C 180,E1 11848.659,E2 11848.659} C_VEL
LIN {X 0,Y 524.682,Z 824.958,A -85,B 0,C 180,E1 11849.956,E2 11849.956} C_VEL
LIN {X 0,Y 529.657,Z 834.387,A -85,B 0,C 180,E1 11851.867,E2 11851.867} C_VEL
LIN {X 0,Y 540.291,Z 857.369,A -85,B 0,C 180,E1 11854.857,E2 11854.857} C_VEL
LIN {X 0,Y 556.294,Z 900.803,A -85,B 0,C 180,E1 11859.554,E2 11859.554} C_VEL
LIN {X 0,Y 559.047,Z 911.721,A -85,B 0,C 180,E1 11860.647,E2 11860.647} C_VEL
LIN {X 0,Y 551.551,Z 950.738,A -85,B 0,C 180,E1 11863.282,E2 11863.282} C_VEL
LIN {X 0,Y 543.274,Z 987.788,A -85,B 0,C 180,E1 11866.53,E2 11866.53} C_VEL
LIN {X 0,Y 535.303,Z 1020.229,A -85,B 0,C 180,E1 11870.249,E2 11870.249} C_VEL
LIN {X 0,Y 527.789,Z 1050,A -85,B 0,C 180,E1 11874.661,E2 11874.661} C_VEL
LIN {X 0,Y 521.339,Z 1081.183,A -85,B 0,C 180,E1 11880.383,E2 11880.383} C_VEL
LIN {X 0,Y 517.593,Z 1103.771,A -85,B 0,C 180,E1 11885.849,E2 11885.849} C_VEL
LIN {X 0,Y 515.984,Z 1118.613,A -85,B 0,C 180,E1 11890.691,E2 11890.691} C_VEL
LIN {X 0,Y 515.007,Z 1130.064,A -85,B 0,C 180,E1 11896.183,E2 11896.183} C_VEL
LIN {X 0,Y 514.455,Z 1135.271,A -85,B 0,C 180,E1 11900.636,E2 11900.636} C_VEL
LIN {X 0,Y 514.201,Z 1136.809,A -85,B 0,C 180,E1 11906.153,E2 11906.153} C_VEL
LIN {X 0,Y 514.801,Z 1132.894,A -85,B 0,C 180,E1 11911.67,E2 11911.67} C_VEL
LIN {X 0,Y 515.474,Z 1124.516,A -85,B 0,C 180,E1 11916.694,E2 11916.694} C_VEL
LIN {X 0,Y 516.764,Z 1111.294,A -85,B 0,C 180,E1 11921.777,E2 11921.777} C_VEL
LIN {X 0,Y 519.503,Z 1092.315,A -85,B 0,C 180,E1 11927.018,E2 11927.018} C_VEL
LIN {X 0,Y 523.909,Z 1067.77,A -85,B 0,C 180,E1 11932.146,E2 11932.146} C_VEL
LIN {X 0,Y 531.485,Z 1033.704,A -85,B 0,C 180,E1 11937.718,E2 11937.718} C_VEL
LIN {X 0,Y 539.713,Z 999.78,A -85,B 0,C 180,E1 11941.968,E2 11941.968} C_VEL
LIN {X 0,Y 548.305,Z 962.211,A -85,B 0,C 180,E1 11945.59,E2 11945.59} C_VEL
LIN {X 0,Y 556.858,Z 921.092,A -85,B 0,C 180,E1 11948.657,E2 11948.657} C_VEL
LIN {X 0,Y 558.761,Z 909.102,A -85,B 0,C 180,E1 11949.424,E2 11949.424} C_VEL
LIN {X 0,Y 546.34,Z 873.675,A -85,B 0,C 180,E1 11953.331,E2 11953.331} C_VEL
LIN {X 0,Y 530.23,Z 839.026,A -85,B 0,C 180,E1 11957.356,E2 11957.356} C_VEL
LIN {X 0,Y 515.969,Z 813.665,A -85,B 0,C 180,E1 11960.525,E2 11960.525} C_VEL
LIN {X 0,Y 514.522,Z 809.06,A -85,B 0,C 180,E1 11961.031,E2 11961.031} C_VEL
LIN {X 0,Y 514.842,Z 809.06,A -85,B 0,C 180,E1 11966.642,E2 11966.642} C_VEL
LIN {X 0,Y 514.831,Z 809.06,A -85,B 0,C 180,E1 11971.689,E2 11971.689} C_VEL
LIN {X 0,Y 514.671,Z 809.06,A -85,B 0,C 180,E1 11976.751,E2 11976.751} C_VEL
LIN {X 0,Y 514.414,Z 809.06,A -85,B 0,C 180,E1 11981.873,E2 11981.873} C_VEL
LIN {X 0,Y 514.276,Z 809.06,A -85,B 0,C 180,E1 11987.094,E2 11987.094} C_VEL
LIN {X 0,Y 514.023,Z 809.06,A -85,B 0,C 180,E1 11992.475,E2 11992.475} C_VEL
LIN {X 0,Y 513.894,Z 809.06,A -85,B 0,C 180,E1 11998.107,E2 11998.107} C_VEL
LIN {X 0,Y 513.716,Z 809.06,A -85,B 0,C 180,E1 12003.986,E2 12003.986} C_VEL
LIN {X 0,Y 513.693,Z 809.06,A -85,B 0,C 180,E1 12010.335,E2 12010.335} C_VEL
LIN {X 0,Y 513.637,Z 809.06,A -85,B 0,C 180,E1 12015.089,E2 12015.089} C_VEL
LIN {X 0,Y 513.635,Z 809.06,A -85,B 0,C 180,E1 12021.847,E2 12021.847} C_VEL
LIN {X 0,Y 513.77,Z 809.06,A -85,B 0,C 180,E1 12028.543,E2 12028.543} C_VEL
LIN {X 0,Y 513.997,Z 809.06,A -85,B 0,C 180,E1 12033.836,E2 12033.836} C_VEL
LIN {X 0,Y 514.145,Z 809.06,A -85,B 0,C 180,E1 12040.15,E2 12040.15} C_VEL
LIN {X 0,Y 514.316,Z 809.06,A -85,B 0,C 180,E1 12046.407,E2 12046.407} C_VEL
LIN {X 0,Y 514.62,Z 809.06,A -85,B 0,C 180,E1 12051.559,E2 12051.559} C_VEL
LIN {X 0,Y 514.805,Z 809.06,A -85,B 0,C 180,E1 12056.635,E2 12056.635} C_VEL
LIN {X 0,Y 514.956,Z 809.06,A -85,B 0,C 180,E1 12061.682,E2 12061.682} C_VEL
LIN {X 0,Y 514.67,Z 809.06,A -85,B 0,C 180,E1 12066.745,E2 12066.745} C_VEL
LIN {X 0,Y 514.421,Z 809.06,A -85,B 0,C 180,E1 12071.866,E2 12071.866} C_VEL
LIN {X 0,Y 514.24,Z 809.06,A -85,B 0,C 180,E1 12077.088,E2 12077.088} C_VEL
LIN {X 0,Y 513.99,Z 809.06,A -85,B 0,C 180,E1 12082.468,E2 12082.468} C_VEL
LIN {X 0,Y 513.851,Z 809.06,A -85,B 0,C 180,E1 12088.078,E2 12088.078} C_VEL
LIN {X 0,Y 513.77,Z 809.318,A -85,B 0,C 180,E1 12090.654,E2 12090.654} C_VEL
LIN {X 0,Y 516.172,Z 814.726,A -85,B 0,C 180,E1 12091.152,E2 12091.152} C_VEL
LIN {X 0,Y 540.223,Z 850.946,A -85,B 0,C 180,E1 12095.255,E2 12095.255} C_VEL
LIN {X 0,Y 565.776,Z 894.169,A -85,B 0,C 180,E1 12099.128,E2 12099.128} C_VEL
LIN {X 0,Y 574.64,Z 912.085,A -85,B 0,C 180,E1 12100.501,E2 12100.501} C_VEL
LIN {X 0,Y 569.367,Z 963.735,A -85,B 0,C 180,E1 12101.802,E2 12101.802} C_VEL
LIN {X 0,Y 562.512,Z 1012.37,A -85,B 0,C 180,E1 12103.696,E2 12103.696} C_VEL
LIN {X 0,Y 554.585,Z 1060.006,A -85,B 0,C 180,E1 12106.252,E2 12106.252} C_VEL
LIN {X 0,Y 545.591,Z 1107.801,A -85,B 0,C 180,E1 12109.679,E2 12109.679} C_VEL
LIN {X 0,Y 537.732,Z 1147.926,A -85,B 0,C 180,E1 12113.393,E2 12113.393} C_VEL
LIN {X 0,Y 530.447,Z 1185.095,A -85,B 0,C 180,E1 12117.708,E2 12117.708} C_VEL
LIN {X 0,Y 525.675,Z 1208.594,A -85,B 0,C 180,E1 12121.186,E2 12121.186} C_VEL
LIN {X 0,Y 525.352,Z 1210.211,A -85,B 0,C 180,E1 12121.453,E2 12121.453} C_VEL
LIN {X 0,Y 519.582,Z 1219.736,A -85,B 0,C 180,E1 12122.945,E2 12122.945} C_VEL
LIN {X 0,Y 514.197,Z 1228.587,A -85,B 0,C 180,E1 12124.514,E2 12124.514} C_VEL
LIN {X 0,Y 510.43,Z 1250.372,A -85,B 0,C 180,E1 12129.637,E2 12129.637} C_VEL
LIN {X 0,Y 508.346,Z 1266.984,A -85,B 0,C 180,E1 12134.924,E2 12134.924} C_VEL
LIN {X 0,Y 507.27,Z 1279.205,A -85,B 0,C 180,E1 12140.564,E2 12140.564} C_VEL
LIN {X 0,Y 507.025,Z 1284.638,A -85,B 0,C 180,E1 12144.864,E2 12144.864} C_VEL
LIN {X 0,Y 507.119,Z 1287,A -85,B 0,C 180,E1 12149.993,E2 12149.993} C_VEL
LIN {X 0,Y 507.014,Z 1284.653,A -85,B 0,C 180,E1 12155.123,E2 12155.123} C_VEL
LIN {X 0,Y 507.358,Z 1277.67,A -85,B 0,C 180,E1 12160.287,E2 12160.287} C_VEL
LIN {X 0,Y 508.428,Z 1265.862,A -85,B 0,C 180,E1 12165.507,E2 12165.507} C_VEL
LIN {X 0,Y 510.707,Z 1248.718,A -85,B 0,C 180,E1 12170.789,E2 12170.789} C_VEL
LIN {X 0,Y 514.771,Z 1225.519,A -85,B 0,C 180,E1 12176.116,E2 12176.116} C_VEL
LIN {X 0,Y 518.921,Z 1205.41,A -85,B 0,C 180,E1 12179.663,E2 12179.663} C_VEL
LIN {X 0,Y 525.172,Z 1171.039,A -85,B 0,C 180,E1 12184.121,E2 12184.121} C_VEL
LIN {X 0,Y 532.105,Z 1132.255,A -85,B 0,C 180,E1 12188.07,E2 12188.07} C_VEL
LIN {X 0,Y 539.567,Z 1088.204,A -85,B 0,C 180,E1 12191.607,E2 12191.607} C_VEL
LIN {X 0,Y 546.72,Z 1041.511,A -85,B 0,C 180,E1 12194.496,E2 12194.496} C_VEL
LIN {X 0,Y 553.742,Z 989.127,A -85,B 0,C 180,E1 12196.949,E2 12196.949} C_VEL
LIN {X 0,Y 560.055,Z 933.027,A -85,B 0,C 180,E1 12198.76,E2 12198.76} C_VEL
LIN {X 0,Y 561.575,Z 912.082,A -85,B 0,C 180,E1 12199.292,E2 12199.292} C_VEL
LIN {X 0,Y 548.406,Z 886.644,A -85,B 0,C 180,E1 12201.184,E2 12201.184} C_VEL
LIN {X 0,Y 534.068,Z 854.62,A -85,B 0,C 180,E1 12203.737,E2 12203.737} C_VEL
LIN {X 0,Y 525.746,Z 838.639,A -85,B 0,C 180,E1 12205.727,E2 12205.727} C_VEL
LIN {X 0,Y 521.987,Z 831.162,A -85,B 0,C 180,E1 12207.377,E2 12207.377} C_VEL
LIN {X 0,Y 521.697,Z 831.038,A -85,B 0,C 180,E1 12209.222,E2 12209.222} C_VEL
LIN {X 0,Y 524.679,Z 837.301,A -85,B 0,C 180,E1 12210.917,E2 12210.917} C_VEL
LIN {X 0,Y 532.839,Z 856.028,A -85,B 0,C 180,E1 12213.697,E2 12213.697} C_VEL
LIN {X 0,Y 547.262,Z 895.668,A -85,B 0,C 180,E1 12218.177,E2 12218.177} C_VEL
LIN {X 0,Y 552.935,Z 914.473,A -85,B 0,C 180,E1 12220.208,E2 12220.208} C_VEL
LIN {X 0,Y 544.936,Z 954.57,A -85,B 0,C 180,E1 12222.969,E2 12222.969} C_VEL
LIN {X 0,Y 536.652,Z 990.255,A -85,B 0,C 180,E1 12226.153,E2 12226.153} C_VEL
LIN {X 0,Y 528.099,Z 1023.998,A -85,B 0,C 180,E1 12230.114,E2 12230.114} C_VEL
LIN {X 0,Y 520.684,Z 1052.208,A -85,B 0,C 180,E1 12234.379,E2 12234.379} C_VEL
LIN {X 0,Y 512.758,Z 1086.702,A -85,B 0,C 180,E1 12241.224,E2 12241.224} C_VEL
LIN {X 0,Y 509.509,Z 1106.402,A -85,B 0,C 180,E1 12246.326,E2 12246.326} C_VEL
LIN {X 0,Y 507.881,Z 1121.017,A -85,B 0,C 180,E1 12251.462,E2 12251.462} C_VEL
LIN {X 0,Y 507.076,Z 1130.633,A -85,B 0,C 180,E1 12256.444,E2 12256.444} C_VEL
LIN {X 0,Y 506.48,Z 1135.592,A -85,B 0,C 180,E1 12260.977,E2 12260.977} C_VEL
LIN {X 0,Y 506.297,Z 1136.737,A -85,B 0,C 180,E1 12266.593,E2 12266.593} C_VEL
LIN {X 0,Y 506.809,Z 1133.424,A -85,B 0,C 180,E1 12271.304,E2 12271.304} C_VEL
LIN {X 0,Y 507.557,Z 1125.277,A -85,B 0,C 180,E1 12276.516,E2 12276.516} C_VEL
LIN {X 0,Y 508.827,Z 1112.524,A -85,B 0,C 180,E1 12281.646,E2 12281.646} C_VEL
LIN {X 0,Y 511.791,Z 1092.837,A -85,B 0,C 180,E1 12287.239,E2 12287.239} C_VEL
LIN {X 0,Y 516.572,Z 1067.792,A -85,B 0,C 180,E1 12292.574,E2 12292.574} C_VEL
LIN {X 0,Y 523.256,Z 1040.07,A -85,B 0,C 180,E1 12297.364,E2 12297.364} C_VEL
LIN {X 0,Y 531.173,Z 1008.355,A -85,B 0,C 180,E1 12301.58,E2 12301.58} C_VEL
LIN {X 0,Y 540.436,Z 970.494,A -85,B 0,C 180,E1 12305.47,E2 12305.47} C_VEL
LIN {X 0,Y 549.431,Z 929.07,A -85,B 0,C 180,E1 12308.707,E2 12308.707} C_VEL
LIN {X 0,Y 552.462,Z 912.471,A -85,B 0,C 180,E1 12309.806,E2 12309.806} C_VEL
LIN {X 0,Y 540.343,Z 877.396,A -85,B 0,C 180,E1 12313.768,E2 12313.768} C_VEL
LIN {X 0,Y 524.392,Z 842.656,A -85,B 0,C 180,E1 12317.902,E2 12317.902} C_VEL
LIN {X 0,Y 508.536,Z 814.145,A -85,B 0,C 180,E1 12321.571,E2 12321.571} C_VEL
LIN {X 0,Y 506.662,Z 809.06,A -85,B 0,C 180,E1 12322.187,E2 12322.187} C_VEL
LIN {X 0,Y 506.881,Z 809.06,A -85,B 0,C 180,E1 12328.299,E2 12328.299} C_VEL
LIN {X 0,Y 506.84,Z 809.06,A -85,B 0,C 180,E1 12333.425,E2 12333.425} C_VEL
LIN {X 0,Y 506.653,Z 809.06,A -85,B 0,C 180,E1 12338.583,E2 12338.583} C_VEL
LIN {X 0,Y 506.478,Z 809.06,A -85,B 0,C 180,E1 12343.816,E2 12343.816} C_VEL
LIN {X 0,Y 506.269,Z 809.06,A -85,B 0,C 180,E1 12349.174,E2 12349.174} C_VEL
LIN {X 0,Y 505.997,Z 809.06,A -85,B 0,C 180,E1 12354.721,E2 12354.721} C_VEL
LIN {X 0,Y 505.882,Z 809.06,A -85,B 0,C 180,E1 12360.524,E2 12360.524} C_VEL
LIN {X 0,Y 505.782,Z 809.06,A -85,B 0,C 180,E1 12366.7,E2 12366.7} C_VEL
LIN {X 0,Y 505.67,Z 809.06,A -85,B 0,C 180,E1 12373.425,E2 12373.425} C_VEL
LIN {X 0,Y 505.634,Z 809.06,A -85,B 0,C 180,E1 12378.897,E2 12378.897} C_VEL
LIN {X 0,Y 505.719,Z 809.06,A -85,B 0,C 180,E1 12385.412,E2 12385.412} C_VEL
LIN {X 0,Y 505.961,Z 809.06,A -85,B 0,C 180,E1 12391.458,E2 12391.458} C_VEL
LIN {X 0,Y 506.187,Z 809.06,A -85,B 0,C 180,E1 12397.746,E2 12397.746} C_VEL
LIN {X 0,Y 506.335,Z 809.06,A -85,B 0,C 180,E1 12402.764,E2 12402.764} C_VEL
LIN {X 0,Y 506.493,Z 809.06,A -85,B 0,C 180,E1 12407.947,E2 12407.947} C_VEL
LIN {X 0,Y 506.756,Z 809.06,A -85,B 0,C 180,E1 12413.151,E2 12413.151} C_VEL
LIN {X 0,Y 506.931,Z 809.06,A -85,B 0,C 180,E1 12418.293,E2 12418.293} C_VEL
LIN {X 0,Y 506.923,Z 809.06,A -85,B 0,C 180,E1 12423.418,E2 12423.418} C_VEL
LIN {X 0,Y 506.667,Z 809.06,A -85,B 0,C 180,E1 12428.576,E2 12428.576} C_VEL
LIN {X 0,Y 506.416,Z 809.06,A -85,B 0,C 180,E1 12433.81,E2 12433.81} C_VEL
LIN {X 0,Y 506.26,Z 809.06,A -85,B 0,C 180,E1 12439.167,E2 12439.167} C_VEL
LIN {X 0,Y 505.968,Z 809.06,A -85,B 0,C 180,E1 12444.715,E2 12444.715} C_VEL
LIN {X 0,Y 505.915,Z 809.784,A -85,B 0,C 180,E1 12449.474,E2 12449.474} C_VEL
LIN {X 0,Y 508.606,Z 814.978,A -85,B 0,C 180,E1 12450.029,E2 12450.029} C_VEL
LIN {X 0,Y 534.646,Z 854.458,A -85,B 0,C 180,E1 12454.634,E2 12454.634} C_VEL
LIN {X 0,Y 560.127,Z 897.356,A -85,B 0,C 180,E1 12458.592,E2 12458.592} C_VEL
LIN {X 0,Y 568.896,Z 914.128,A -85,B 0,C 180,E1 12459.978,E2 12459.978} C_VEL
LIN {X 0,Y 563.518,Z 963.977,A -85,B 0,C 180,E1 12461.264,E2 12461.264} C_VEL
LIN {X 0,Y 556.16,Z 1013.972,A -85,B 0,C 180,E1 12463.24,E2 12463.24} C_VEL
LIN {X 0,Y 548.363,Z 1059.138,A -85,B 0,C 180,E1 12465.701,E2 12465.701} C_VEL
LIN {X 0,Y 539.154,Z 1106.271,A -85,B 0,C 180,E1 12469.107,E2 12469.107} C_VEL
LIN {X 0,Y 530.842,Z 1146.44,A -85,B 0,C 180,E1 12472.845,E2 12472.845} C_VEL
LIN {X 0,Y 522.916,Z 1185.36,A -85,B 0,C 180,E1 12477.431,E2 12477.431} C_VEL
LIN {X 0,Y 517.063,Z 1214.742,A -85,B 0,C 180,E1 12481.835,E2 12481.835} C_VEL
LIN {X 0,Y 514.197,Z 1228.587,A -85,B 0,C 180,E1 12484.514,E2 12484.514} C_VEL
LIN {X 0,Y 508.959,Z 1236.945,A -85,B 0,C 180,E1 12486.138,E2 12486.138} C_VEL
LIN {X 0,Y 503.717,Z 1244.665,A -85,B 0,C 180,E1 12487.827,E2 12487.827} C_VEL
LIN {X 0,Y 500.909,Z 1263.346,A -85,B 0,C 180,E1 12493.339,E2 12493.339} C_VEL
LIN {X 0,Y 499.629,Z 1276.08,A -85,B 0,C 180,E1 12498.656,E2 12498.656} C_VEL
LIN {X 0,Y 499.274,Z 1282.901,A -85,B 0,C 180,E1 12503.04,E2 12503.04} C_VEL
LIN {X 0,Y 499.09,Z 1286.664,A -85,B 0,C 180,E1 12508.258,E2 12508.258} C_VEL
LIN {X 0,Y 499.195,Z 1286.317,A -85,B 0,C 180,E1 12512.721,E2 12512.721} C_VEL
LIN {X 0,Y 499.287,Z 1281.745,A -85,B 0,C 180,E1 12517.82,E2 12517.82} C_VEL
LIN {X 0,Y 500.002,Z 1272.378,A -85,B 0,C 180,E1 12523.093,E2 12523.093} C_VEL
LIN {X 0,Y 501.844,Z 1257.237,A -85,B 0,C 180,E1 12528.673,E2 12528.673} C_VEL
LIN {X 0,Y 505.568,Z 1235.528,A -85,B 0,C 180,E1 12534.36,E2 12534.36} C_VEL
LIN {X 0,Y 508.914,Z 1217.482,A -85,B 0,C 180,E1 12537.901,E2 12537.901} C_VEL
LIN {X 0,Y 514.895,Z 1185.303,A -85,B 0,C 180,E1 12542.586,E2 12542.586} C_VEL
LIN {X 0,Y 521.707,Z 1148.483,A -85,B 0,C 180,E1 12546.803,E2 12546.803} C_VEL
LIN {X 0,Y 529.327,Z 1105.987,A -85,B 0,C 180,E1 12550.624,E2 12550.624} C_VEL
LIN {X 0,Y 536.698,Z 1062.264,A -85,B 0,C 180,E1 12553.697,E2 12553.697} C_VEL
LIN {X 0,Y 544.239,Z 1011.703,A -85,B 0,C 180,E1 12556.415,E2 12556.415} C_VEL
LIN {X 0,Y 550.527,Z 962.918,A -85,B 0,C 180,E1 12558.358,E2 12558.358} C_VEL
LIN {X 0,Y 555.03,Z 915.164,A -85,B 0,C 180,E1 12559.746,E2 12559.746} C_VEL
LIN {X 0,Y 542.997,Z 890.655,A -85,B 0,C 180,E1 12561.618,E2 12561.618} C_VEL
LIN {X 0,Y 530.286,Z 860.885,A -85,B 0,C 180,E1 12564.088,E2 12564.088} C_VEL
LIN {X 0,Y 523.128,Z 845.919,A -85,B 0,C 180,E1 12565.97,E2 12565.97} C_VEL
LIN {X 0,Y 519.961,Z 838.662,A -85,B 0,C 180,E1 12567.621,E2 12567.621} C_VEL
LIN {X 0,Y 519.851,Z 839.081,A -85,B 0,C 180,E1 12569.358,E2 12569.358} C_VEL
LIN {X 0,Y 523.383,Z 848.722,A -85,B 0,C 180,E1 12571.455,E2 12571.455} C_VEL
LIN {X 0,Y 532.953,Z 873.863,A -85,B 0,C 180,E1 12574.832,E2 12574.832} C_VEL
LIN {X 0,Y 546.9,Z 916.74,A -85,B 0,C 180,E1 12579.717,E2 12579.717} C_VEL
LIN {X 0,Y 538.606,Z 957.239,A -85,B 0,C 180,E1 12582.552,E2 12582.552} C_VEL
LIN {X 0,Y 530.06,Z 992.716,A -85,B 0,C 180,E1 12585.766,E2 12585.766} C_VEL
LIN {X 0,Y 521.229,Z 1026.302,A -85,B 0,C 180,E1 12589.772,E2 12589.772} C_VEL
LIN {X 0,Y 513.585,Z 1054.419,A -85,B 0,C 180,E1 12594.089,E2 12594.089} C_VEL
LIN {X 0,Y 507.031,Z 1078.868,A -85,B 0,C 180,E1 12599.016,E2 12599.016} C_VEL
LIN {X 0,Y 502.252,Z 1103.557,A -85,B 0,C 180,E1 12605.177,E2 12605.177} C_VEL
LIN {X 0,Y 500.268,Z 1119.117,A -85,B 0,C 180,E1 12610.44,E2 12610.44} C_VEL
LIN {X 0,Y 499.242,Z 1129.92,A -85,B 0,C 180,E1 12615.806,E2 12615.806} C_VEL
LIN {X 0,Y 498.654,Z 1134.936,A -85,B 0,C 180,E1 12620.074,E2 12620.074} C_VEL
LIN {X 0,Y 498.336,Z 1136.979,A -85,B 0,C 180,E1 12625.118,E2 12625.118} C_VEL
LIN {X 0,Y 498.562,Z 1135.587,A -85,B 0,C 180,E1 12629.006,E2 12629.006} C_VEL
LIN {X 0,Y 499.325,Z 1129.95,A -85,B 0,C 180,E1 12634.072,E2 12634.072} C_VEL
LIN {X 0,Y 500.333,Z 1119.347,A -85,B 0,C 180,E1 12639.359,E2 12639.359} C_VEL
LIN {X 0,Y 502.484,Z 1102.415,A -85,B 0,C 180,E1 12645.058,E2 12645.058} C_VEL
LIN {X 0,Y 507.131,Z 1077.916,A -85,B 0,C 180,E1 12651.054,E2 12651.054} C_VEL
LIN {X 0,Y 513.469,Z 1052.258,A -85,B 0,C 180,E1 12656.012,E2 12656.012} C_VEL
LIN {X 0,Y 521.294,Z 1022.002,A -85,B 0,C 180,E1 12660.485,E2 12660.485} C_VEL
LIN {X 0,Y 530.371,Z 987.16,A -85,B 0,C 180,E1 12664.484,E2 12664.484} C_VEL
LIN {X 0,Y 539.464,Z 948.686,A -85,B 0,C 180,E1 12667.876,E2 12667.876} C_VEL
LIN {X 0,Y 546.074,Z 915.476,A -85,B 0,C 180,E1 12670.234,E2 12670.234} C_VEL
LIN {X 0,Y 534.351,Z 881.055,A -85,B 0,C 180,E1 12674.214,E2 12674.214} C_VEL
LIN {X 0,Y 519.387,Z 847.907,A -85,B 0,C 180,E1 12678.256,E2 12678.256} C_VEL
LIN {X 0,Y 503.921,Z 819.569,A -85,B 0,C 180,E1 12682.004,E2 12682.004} C_VEL
LIN {X 0,Y 498.934,Z 810.092,A -85,B 0,C 180,E1 12683.213,E2 12683.213} C_VEL
LIN {X 0,Y 498.85,Z 809.06,A -85,B 0,C 180,E1 12683.485,E2 12683.485} C_VEL
LIN {X 0,Y 498.994,Z 809.06,A -85,B 0,C 180,E1 12688.272,E2 12688.272} C_VEL
LIN {X 0,Y 498.945,Z 809.06,A -85,B 0,C 180,E1 12693.48,E2 12693.48} C_VEL
LIN {X 0,Y 498.735,Z 809.06,A -85,B 0,C 180,E1 12698.72,E2 12698.72} C_VEL
LIN {X 0,Y 498.542,Z 809.06,A -85,B 0,C 180,E1 12704.105,E2 12704.105} C_VEL
LIN {X 0,Y 498.262,Z 809.06,A -85,B 0,C 180,E1 12709.937,E2 12709.937} C_VEL
LIN {X 0,Y 498.08,Z 809.06,A -85,B 0,C 180,E1 12715.141,E2 12715.141} C_VEL
LIN {X 0,Y 497.902,Z 809.06,A -85,B 0,C 180,E1 12721.067,E2 12721.067} C_VEL
LIN {X 0,Y 497.786,Z 809.06,A -85,B 0,C 180,E1 12727.389,E2 12727.389} C_VEL
LIN {X 0,Y 497.765,Z 809.06,A -85,B 0,C 180,E1 12733.238,E2 12733.238} C_VEL
LIN {X 0,Y 497.695,Z 809.06,A -85,B 0,C 180,E1 12739.389,E2 12739.389} C_VEL
LIN {X 0,Y 497.81,Z 809.06,A -85,B 0,C 180,E1 12745.053,E2 12745.053} C_VEL
LIN {X 0,Y 498.057,Z 809.06,A -85,B 0,C 180,E1 12751.636,E2 12751.636} C_VEL
LIN {X 0,Y 498.167,Z 809.06,A -85,B 0,C 180,E1 12756.778,E2 12756.778} C_VEL
LIN {X 0,Y 498.372,Z 809.06,A -85,B 0,C 180,E1 12762.352,E2 12762.352} C_VEL
LIN {X 0,Y 498.559,Z 809.06,A -85,B 0,C 180,E1 12767.752,E2 12767.752} C_VEL
LIN {X 0,Y 498.83,Z 809.06,A -85,B 0,C 180,E1 12773.143,E2 12773.143} C_VEL
LIN {X 0,Y 499.036,Z 809.06,A -85,B 0,C 180,E1 12778.266,E2 12778.266} C_VEL
LIN {X 0,Y 499.026,Z 809.06,A -85,B 0,C 180,E1 12783.472,E2 12783.472} C_VEL
LIN {X 0,Y 498.75,Z 809.06,A -85,B 0,C 180,E1 12788.713,E2 12788.713} C_VEL
LIN {X 0,Y 498.496,Z 809.06,A -85,B 0,C 180,E1 12794.044,E2 12794.044} C_VEL
LIN {X 0,Y 498.249,Z 809.06,A -85,B 0,C 180,E1 12799.904,E2 12799.904} C_VEL
LIN {X 0,Y 498.059,Z 809.06,A -85,B 0,C 180,E1 12805.134,E2 12805.134} C_VEL
LIN {X 0,Y 497.985,Z 809.06,A -85,B 0,C 180,E1 12808.204,E2 12808.204} C_VEL
LIN {X 0,Y 500.175,Z 814.509,A -85,B 0,C 180,E1 12808.715,E2 12808.715} C_VEL
LIN {X 0,Y 514.959,Z 836.141,A -85,B 0,C 180,E1 12811.531,E2 12811.531} C_VEL
LIN {X 0,Y 540.054,Z 875.495,A -85,B 0,C 180,E1 12815.77,E2 12815.77} C_VEL
LIN {X 0,Y 561.29,Z 914.157,A -85,B 0,C 180,E1 12819.182,E2 12819.182} C_VEL
LIN {X 0,Y 563.04,Z 918.765,A -85,B 0,C 180,E1 12819.503,E2 12819.503} C_VEL
LIN {X 0,Y 557.014,Z 968.627,A -85,B 0,C 180,E1 12820.862,E2 12820.862} C_VEL
LIN {X 0,Y 549.391,Z 1018.541,A -85,B 0,C 180,E1 12822.919,E2 12822.919} C_VEL
LIN {X 0,Y 540.536,Z 1066.247,A -85,B 0,C 180,E1 12825.655,E2 12825.655} C_VEL
LIN {X 0,Y 531.6,Z 1109.768,A -85,B 0,C 180,E1 12828.929,E2 12828.929} C_VEL
LIN {X 0,Y 522.426,Z 1152.6,A -85,B 0,C 180,E1 12833.11,E2 12833.11} C_VEL
LIN {X 0,Y 515.026,Z 1187.356,A -85,B 0,C 180,E1 12837.405,E2 12837.405} C_VEL
LIN {X 0,Y 508.508,Z 1220.084,A -85,B 0,C 180,E1 12842.512,E2 12842.512} C_VEL
LIN {X 0,Y 504.582,Z 1240.204,A -85,B 0,C 180,E1 12846.716,E2 12846.716} C_VEL
LIN {X 0,Y 503.717,Z 1244.665,A -85,B 0,C 180,E1 12847.827,E2 12847.827} C_VEL
LIN {X 0,Y 498.709,Z 1251.803,A -85,B 0,C 180,E1 12849.569,E2 12849.569} C_VEL
LIN {X 0,Y 493.922,Z 1258.305,A -85,B 0,C 180,E1 12851.368,E2 12851.368} C_VEL
LIN {X 0,Y 492.065,Z 1272.345,A -85,B 0,C 180,E1 12856.677,E2 12856.677} C_VEL
LIN {X 0,Y 491.388,Z 1281.721,A -85,B 0,C 180,E1 12862.039,E2 12862.039} C_VEL
LIN {X 0,Y 491.248,Z 1285.869,A -85,B 0,C 180,E1 12866.466,E2 12866.466} C_VEL
LIN {X 0,Y 491.411,Z 1286.667,A -85,B 0,C 180,E1 12871.755,E2 12871.755} C_VEL
LIN {X 0,Y 491.362,Z 1282.919,A -85,B 0,C 180,E1 12877.059,E2 12877.059} C_VEL
LIN {X 0,Y 491.957,Z 1274.297,A -85,B 0,C 180,E1 12882.408,E2 12882.408} C_VEL
LIN {X 0,Y 493.469,Z 1260.723,A -85,B 0,C 180,E1 12887.823,E2 12887.823} C_VEL
LIN {X 0,Y 496.739,Z 1241.764,A -85,B 0,C 180,E1 12893.286,E2 12893.286} C_VEL
LIN {X 0,Y 500.568,Z 1220.317,A -85,B 0,C 180,E1 12897.526,E2 12897.526} C_VEL
LIN {X 0,Y 506.434,Z 1188.929,A -85,B 0,C 180,E1 12902.288,E2 12902.288} C_VEL
LIN {X 0,Y 513.523,Z 1152.308,A -85,B 0,C 180,E1 12906.687,E2 12906.687} C_VEL
LIN {X 0,Y 520.838,Z 1112.513,A -85,B 0,C 180,E1 12910.437,E2 12910.437} C_VEL
LIN {X 0,Y 529.111,Z 1066.011,A -85,B 0,C 180,E1 12913.862,E2 12913.862} C_VEL
LIN {X 0,Y 536.568,Z 1018.931,A -85,B 0,C 180,E1 12916.517,E2 12916.517} C_VEL
LIN {X 0,Y 543.22,Z 970.12,A -85,B 0,C 180,E1 12918.591,E2 12918.591} C_VEL
LIN {X 0,Y 548.771,Z 918.6,A -85,B 0,C 180,E1 12920.185,E2 12920.185} C_VEL
LIN {X 0,Y 537.325,Z 893.879,A -85,B 0,C 180,E1 12922.121,E2 12922.121} C_VEL
LIN {X 0,Y 525.433,Z 864.551,A -85,B 0,C 180,E1 12924.693,E2 12924.693} C_VEL
LIN {X 0,Y 519.402,Z 850.254,A -85,B 0,C 180,E1 12926.712,E2 12926.712} C_VEL
LIN {X 0,Y 517.895,Z 846.227,A -85,B 0,C 180,E1 12927.78,E2 12927.78} C_VEL
LIN {X 0,Y 517.645,Z 846.879,A -85,B 0,C 180,E1 12929.22,E2 12929.22} C_VEL
LIN {X 0,Y 519.971,Z 855.035,A -85,B 0,C 180,E1 12931.086,E2 12931.086} C_VEL
LIN {X 0,Y 527.487,Z 876.898,A -85,B 0,C 180,E1 12934.201,E2 12934.201} C_VEL
LIN {X 0,Y 540.638,Z 919.669,A -85,B 0,C 180,E1 12939.231,E2 12939.231} C_VEL
LIN {X 0,Y 531.759,Z 962.371,A -85,B 0,C 180,E1 12942.32,E2 12942.32} C_VEL
LIN {X 0,Y 523.027,Z 996.997,A -85,B 0,C 180,E1 12945.571,E2 12945.571} C_VEL
LIN {X 0,Y 513.543,Z 1031.649,A -85,B 0,C 180,E1 12949.831,E2 12949.831} C_VEL
LIN {X 0,Y 505.414,Z 1060.02,A -85,B 0,C 180,E1 12954.424,E2 12954.424} C_VEL
LIN {X 0,Y 498.828,Z 1084.358,A -85,B 0,C 180,E1 12959.603,E2 12959.603} C_VEL
LIN {X 0,Y 493.742,Z 1108.688,A -85,B 0,C 180,E1 12966.428,E2 12966.428} C_VEL
LIN {X 0,Y 492.094,Z 1122.242,A -85,B 0,C 180,E1 12971.553,E2 12971.553} C_VEL
LIN {X 0,Y 491.245,Z 1131.504,A -85,B 0,C 180,E1 12976.8,E2 12976.8} C_VEL
LIN {X 0,Y 490.553,Z 1136.084,A -85,B 0,C 180,E1 12981.692,E2 12981.692} C_VEL
LIN {X 0,Y 490.499,Z 1136.404,A -85,B 0,C 180,E1 12987.52,E2 12987.52} C_VEL
LIN {X 0,Y 491.192,Z 1132.204,A -85,B 0,C 180,E1 12992.607,E2 12992.607} C_VEL
LIN {X 0,Y 492.098,Z 1123.243,A -85,B 0,C 180,E1 12997.886,E2 12997.886} C_VEL
LIN {X 0,Y 493.916,Z 1108.27,A -85,B 0,C 180,E1 13003.603,E2 13003.603} C_VEL
LIN {X 0,Y 498.883,Z 1082.972,A -85,B 0,C 180,E1 13010.511,E2 13010.511} C_VEL
LIN {X 0,Y 505.305,Z 1057.564,A -85,B 0,C 180,E1 13015.695,E2 13015.695} C_VEL
LIN {X 0,Y 513.429,Z 1027.514,A -85,B 0,C 180,E1 13020.37,E2 13020.37} C_VEL
LIN {X 0,Y 522.603,Z 993.232,A -85,B 0,C 180,E1 13024.461,E2 13024.461} C_VEL
LIN {X 0,Y 532.07,Z 955.621,A -85,B 0,C 180,E1 13027.947,E2 13027.947} C_VEL
LIN {X 0,Y 539.626,Z 918.348,A -85,B 0,C 180,E1 13030.691,E2 13030.691} C_VEL
LIN {X 0,Y 528.333,Z 884.596,A -85,B 0,C 180,E1 13034.685,E2 13034.685} C_VEL
LIN {X 0,Y 513.149,Z 850.354,A -85,B 0,C 180,E1 13038.961,E2 13038.961} C_VEL
LIN {X 0,Y 496.619,Z 820.355,A -85,B 0,C 180,E1 13043.071,E2 13043.071} C_VEL
LIN {X 0,Y 492.677,Z 813.975,A -85,B 0,C 180,E1 13044.011,E2 13044.011} C_VEL
LIN {X 0,Y 491.041,Z 809.06,A -85,B 0,C 180,E1 13044.6,E2 13044.6} C_VEL
LIN {X 0,Y 491.285,Z 809.06,A -85,B 0,C 180,E1 13050.007,E2 13050.007} C_VEL
LIN {X 0,Y 491.038,Z 809.06,A -85,B 0,C 180,E1 13055.304,E2 13055.304} C_VEL
LIN {X 0,Y 490.748,Z 809.06,A -85,B 0,C 180,E1 13060.654,E2 13060.654} C_VEL
LIN {X 0,Y 490.518,Z 809.06,A -85,B 0,C 180,E1 13066.103,E2 13066.103} C_VEL
LIN {X 0,Y 490.2,Z 809.06,A -85,B 0,C 180,E1 13072.376,E2 13072.376} C_VEL
LIN {X 0,Y 490.117,Z 809.06,A -85,B 0,C 180,E1 13077.554,E2 13077.554} C_VEL
LIN {X 0,Y 489.954,Z 809.06,A -85,B 0,C 180,E1 13083.728,E2 13083.728} C_VEL
LIN {X 0,Y 489.849,Z 809.06,A -85,B 0,C 180,E1 13090.385,E2 13090.385} C_VEL
LIN {X 0,Y 489.835,Z 809.06,A -85,B 0,C 180,E1 13095.205,E2 13095.205} C_VEL
LIN {X 0,Y 489.785,Z 809.06,A -85,B 0,C 180,E1 13100.48,E2 13100.48} C_VEL
LIN {X 0,Y 489.877,Z 809.06,A -85,B 0,C 180,E1 13106.403,E2 13106.403} C_VEL
LIN {X 0,Y 490.15,Z 809.06,A -85,B 0,C 180,E1 13112.458,E2 13112.458} C_VEL
LIN {X 0,Y 490.312,Z 809.06,A -85,B 0,C 180,E1 13118.297,E2 13118.297} C_VEL
LIN {X 0,Y 490.477,Z 809.06,A -85,B 0,C 180,E1 13123.904,E2 13123.904} C_VEL
LIN {X 0,Y 490.761,Z 809.06,A -85,B 0,C 180,E1 13130.197,E2 13130.197} C_VEL
LIN {X 0,Y 491.115,Z 809.06,A -85,B 0,C 180,E1 13136.473,E2 13136.473} C_VEL
LIN {X 0,Y 491.277,Z 809.06,A -85,B 0,C 180,E1 13141.763,E2 13141.763} C_VEL
LIN {X 0,Y 490.912,Z 809.06,A -85,B 0,C 180,E1 13147.073,E2 13147.073} C_VEL
LIN {X 0,Y 490.646,Z 809.06,A -85,B 0,C 180,E1 13152.45,E2 13152.45} C_VEL
LIN {X 0,Y 490.428,Z 809.06,A -85,B 0,C 180,E1 13157.945,E2 13157.945} C_VEL
LIN {X 0,Y 490.161,Z 809.06,A -85,B 0,C 180,E1 13163.625,E2 13163.625} C_VEL
LIN {X 0,Y 490.112,Z 809.46,A -85,B 0,C 180,E1 13166.913,E2 13166.913} C_VEL
LIN {X 0,Y 492.666,Z 814.877,A -85,B 0,C 180,E1 13167.505,E2 13167.505} C_VEL
LIN {X 0,Y 516.912,Z 850.872,A -85,B 0,C 180,E1 13172.186,E2 13172.186} C_VEL
LIN {X 0,Y 542.486,Z 892.6,A -85,B 0,C 180,E1 13176.477,E2 13176.477} C_VEL
LIN {X 0,Y 557.321,Z 921.534,A -85,B 0,C 180,E1 13178.983,E2 13178.983} C_VEL
LIN {X 0,Y 550.535,Z 973.432,A -85,B 0,C 180,E1 13180.457,E2 13180.457} C_VEL
LIN {X 0,Y 542.985,Z 1020.521,A -85,B 0,C 180,E1 13182.475,E2 13182.475} C_VEL
LIN {X 0,Y 533.554,Z 1069.271,A -85,B 0,C 180,E1 13185.347,E2 13185.347} C_VEL
LIN {X 0,Y 524.525,Z 1111.089,A -85,B 0,C 180,E1 13188.579,E2 13188.579} C_VEL
LIN {X 0,Y 515,Z 1153.861,A -85,B 0,C 180,E1 13192.844,E2 13192.844} C_VEL
LIN {X 0,Y 506.886,Z 1190.459,A -85,B 0,C 180,E1 13197.54,E2 13197.54} C_VEL
LIN {X 0,Y 500.617,Z 1220.95,A -85,B 0,C 180,E1 13202.46,E2 13202.46} C_VEL
LIN {X 0,Y 496.356,Z 1243.464,A -85,B 0,C 180,E1 13207.153,E2 13207.153} C_VEL
LIN {X 0,Y 493.922,Z 1258.305,A -85,B 0,C 180,E1 13211.368,E2 13211.368} C_VEL
LIN {X 0,Y 489.304,Z 1264.169,A -85,B 0,C 180,E1 13213.218,E2 13213.218} C_VEL
LIN {X 0,Y 484.674,Z 1269.33,A -85,B 0,C 180,E1 13215.119,E2 13215.119} C_VEL
LIN {X 0,Y 483.635,Z 1279.571,A -85,B 0,C 180,E1 13220.321,E2 13220.321} C_VEL
LIN {X 0,Y 483.371,Z 1284.63,A -85,B 0,C 180,E1 13224.611,E2 13224.611} C_VEL
LIN {X 0,Y 483.435,Z 1287,A -85,B 0,C 180,E1 13229.993,E2 13229.993} C_VEL
LIN {X 0,Y 483.36,Z 1284.645,A -85,B 0,C 180,E1 13235.374,E2 13235.374} C_VEL
LIN {X 0,Y 483.781,Z 1277.661,A -85,B 0,C 180,E1 13240.794,E2 13240.794} C_VEL
LIN {X 0,Y 485.022,Z 1265.86,A -85,B 0,C 180,E1 13246.276,E2 13246.276} C_VEL
LIN {X 0,Y 487.394,Z 1250.741,A -85,B 0,C 180,E1 13251.219,E2 13251.219} C_VEL
LIN {X 0,Y 490.918,Z 1229.392,A -85,B 0,C 180,E1 13255.921,E2 13255.921} C_VEL
LIN {X 0,Y 496.401,Z 1200.626,A -85,B 0,C 180,E1 13260.793,E2 13260.793} C_VEL
LIN {X 0,Y 503.261,Z 1165.921,A -85,B 0,C 180,E1 13265.431,E2 13265.431} C_VEL
LIN {X 0,Y 510.974,Z 1126.755,A -85,B 0,C 180,E1 13269.514,E2 13269.514} C_VEL
LIN {X 0,Y 519.425,Z 1081.533,A -85,B 0,C 180,E1 13273.211,E2 13273.211} C_VEL
LIN {X 0,Y 527.437,Z 1034.1,A -85,B 0,C 180,E1 13276.186,E2 13276.186} C_VEL
LIN {X 0,Y 535.31,Z 981.651,A -85,B 0,C 180,E1 13278.661,E2 13278.661} C_VEL
LIN {X 0,Y 542.373,Z 926.005,A -85,B 0,C 180,E1 13280.488,E2 13280.488} C_VEL
LIN {X 0,Y 542.064,Z 921.155,A -85,B 0,C 180,E1 13280.7,E2 13280.7} C_VEL
LIN {X 0,Y 529.226,Z 890.67,A -85,B 0,C 180,E1 13283.16,E2 13283.16} C_VEL
LIN {X 0,Y 520.167,Z 866.967,A -85,B 0,C 180,E1 13285.512,E2 13285.512} C_VEL
LIN {X 0,Y 516.251,Z 856.036,A -85,B 0,C 180,E1 13287.304,E2 13287.304} C_VEL
LIN {X 0,Y 515.557,Z 853.666,A -85,B 0,C 180,E1 13288.194,E2 13288.194} C_VEL
LIN {X 0,Y 515.336,Z 854.889,A -85,B 0,C 180,E1 13289.151,E2 13289.151} C_VEL
LIN {X 0,Y 517.008,Z 863.043,A -85,B 0,C 180,E1 13291.012,E2 13291.012} C_VEL
LIN {X 0,Y 524.359,Z 887.805,A -85,B 0,C 180,E1 13294.512,E2 13294.512} C_VEL
LIN {X 0,Y 534.534,Z 924.338,A -85,B 0,C 180,E1 13298.901,E2 13298.901} C_VEL
LIN {X 0,Y 525.769,Z 963.963,A -85,B 0,C 180,E1 13301.787,E2 13301.787} C_VEL
LIN {X 0,Y 516.982,Z 997.709,A -85,B 0,C 180,E1 13304.965,E2 13304.965} C_VEL
LIN {X 0,Y 507.14,Z 1032.447,A -85,B 0,C 180,E1 13309.267,E2 13309.267} C_VEL
LIN {X 0,Y 499.002,Z 1059.899,A -85,B 0,C 180,E1 13313.698,E2 13313.698} C_VEL
LIN {X 0,Y 492.166,Z 1083.679,A -85,B 0,C 180,E1 13318.717,E2 13318.717} C_VEL
LIN {X 0,Y 487.024,Z 1103.855,A -85,B 0,C 180,E1 13324.448,E2 13324.448} C_VEL
LIN {X 0,Y 484.39,Z 1120.995,A -85,B 0,C 180,E1 13330.787,E2 13330.787} C_VEL
LIN {X 0,Y 483.517,Z 1129.772,A -85,B 0,C 180,E1 13335.403,E2 13335.403} C_VEL
LIN {X 0,Y 482.829,Z 1135.117,A -85,B 0,C 180,E1 13340.159,E2 13340.159} C_VEL
LIN {X 0,Y 482.49,Z 1136.844,A -85,B 0,C 180,E1 13346.003,E2 13346.003} C_VEL
LIN {X 0,Y 482.997,Z 1134.063,A -85,B 0,C 180,E1 13351.018,E2 13351.018} C_VEL
LIN {X 0,Y 483.929,Z 1126.618,A -85,B 0,C 180,E1 13356.387,E2 13356.387} C_VEL
LIN {X 0,Y 485.188,Z 1114.77,A -85,B 0,C 180,E1 13361.642,E2 13361.642} C_VEL
LIN {X 0,Y 489.269,Z 1093.74,A -85,B 0,C 180,E1 13368.394,E2 13368.394} C_VEL
LIN {X 0,Y 495.006,Z 1070.929,A -85,B 0,C 180,E1 13373.759,E2 13373.759} C_VEL
LIN {X 0,Y 502.571,Z 1043.372,A -85,B 0,C 180,E1 13378.684,E2 13378.684} C_VEL
LIN {X 0,Y 511.443,Z 1011.418,A -85,B 0,C 180,E1 13383.048,E2 13383.048} C_VEL
LIN {X 0,Y 521.474,Z 974.341,A -85,B 0,C 180,E1 13386.965,E2 13386.965} C_VEL
LIN {X 0,Y 531.371,Z 932.888,A -85,B 0,C 180,E1 13390.288,E2 13390.288} C_VEL
LIN {X 0,Y 533.581,Z 922.581,A -85,B 0,C 180,E1 13391.001,E2 13391.001} C_VEL
LIN {X 0,Y 523.069,Z 890.036,A -85,B 0,C 180,E1 13394.937,E2 13394.937} C_VEL
LIN {X 0,Y 508.283,Z 855.837,A -85,B 0,C 180,E1 13399.294,E2 13399.294} C_VEL
LIN {X 0,Y 492.218,Z 826.02,A -85,B 0,C 180,E1 13403.474,E2 13403.474} C_VEL
LIN {X 0,Y 484.857,Z 813.952,A -85,B 0,C 180,E1 13405.299,E2 13405.299} C_VEL
LIN {X 0,Y 483.19,Z 809.06,A -85,B 0,C 180,E1 13405.916,E2 13405.916} C_VEL
LIN {X 0,Y 483.25,Z 809.06,A -85,B 0,C 180,E1 13411.799,E2 13411.799} C_VEL
LIN {X 0,Y 482.991,Z 809.06,A -85,B 0,C 180,E1 13417.196,E2 13417.196} C_VEL
LIN {X 0,Y 482.723,Z 809.06,A -85,B 0,C 180,E1 13422.665,E2 13422.665} C_VEL
LIN {X 0,Y 482.519,Z 809.06,A -85,B 0,C 180,E1 13428.257,E2 13428.257} C_VEL
LIN {X 0,Y 482.187,Z 809.06,A -85,B 0,C 180,E1 13434.669,E2 13434.669} C_VEL
LIN {X 0,Y 482.11,Z 809.06,A -85,B 0,C 180,E1 13440.106,E2 13440.106} C_VEL
LIN {X 0,Y 481.96,Z 809.06,A -85,B 0,C 180,E1 13446.571,E2 13446.571} C_VEL
LIN {X 0,Y 481.905,Z 809.06,A -85,B 0,C 180,E1 13451.193,E2 13451.193} C_VEL
LIN {X 0,Y 481.851,Z 809.06,A -85,B 0,C 180,E1 13456.381,E2 13456.381} C_VEL
LIN {X 0,Y 481.879,Z 809.06,A -85,B 0,C 180,E1 13461.634,E2 13461.634} C_VEL
LIN {X 0,Y 481.992,Z 809.06,A -85,B 0,C 180,E1 13467.841,E2 13467.841} C_VEL
LIN {X 0,Y 482.256,Z 809.06,A -85,B 0,C 180,E1 13473.983,E2 13473.983} C_VEL
LIN {X 0,Y 482.495,Z 809.06,A -85,B 0,C 180,E1 13479.992,E2 13479.992} C_VEL
LIN {X 0,Y 482.631,Z 809.06,A -85,B 0,C 180,E1 13486.094,E2 13486.094} C_VEL
LIN {X 0,Y 482.952,Z 809.06,A -85,B 0,C 180,E1 13491.001,E2 13491.001} C_VEL
LIN {X 0,Y 483.214,Z 809.06,A -85,B 0,C 180,E1 13496.415,E2 13496.415} C_VEL
LIN {X 0,Y 483.385,Z 809.06,A -85,B 0,C 180,E1 13501.792,E2 13501.792} C_VEL
LIN {X 0,Y 482.999,Z 809.06,A -85,B 0,C 180,E1 13507.189,E2 13507.189} C_VEL
LIN {X 0,Y 482.714,Z 809.06,A -85,B 0,C 180,E1 13512.658,E2 13512.658} C_VEL
LIN {X 0,Y 482.483,Z 809.06,A -85,B 0,C 180,E1 13518.251,E2 13518.251} C_VEL
LIN {X 0,Y 482.169,Z 809.06,A -85,B 0,C 180,E1 13524.64,E2 13524.64} C_VEL
LIN {X 0,Y 482.234,Z 809.482,A -85,B 0,C 180,E1 13525.559,E2 13525.559} C_VEL
LIN {X 0,Y 484.6,Z 814.766,A -85,B 0,C 180,E1 13526.138,E2 13526.138} C_VEL
LIN {X 0,Y 503.714,Z 842.49,A -85,B 0,C 180,E1 13530.039,E2 13530.039} C_VEL
LIN {X 0,Y 528.845,Z 882.124,A -85,B 0,C 180,E1 13534.54,E2 13534.54} C_VEL
LIN {X 0,Y 548.665,Z 918.716,A -85,B 0,C 180,E1 13537.96,E2 13537.96} C_VEL
LIN {X 0,Y 551.421,Z 924.259,A -85,B 0,C 180,E1 13538.458,E2 13538.458} C_VEL
LIN {X 0,Y 544.283,Z 976.987,A -85,B 0,C 180,E1 13540.012,E2 13540.012} C_VEL
LIN {X 0,Y 536.435,Z 1023.373,A -85,B 0,C 180,E1 13542.074,E2 13542.074} C_VEL
LIN {X 0,Y 526.732,Z 1071.415,A -85,B 0,C 180,E1 13544.969,E2 13544.969} C_VEL
LIN {X 0,Y 516.731,Z 1115.383,A -85,B 0,C 180,E1 13548.488,E2 13548.488} C_VEL
LIN {X 0,Y 507.657,Z 1154.685,A -85,B 0,C 180,E1 13552.53,E2 13552.53} C_VEL
LIN {X 0,Y 498.973,Z 1192.282,A -85,B 0,C 180,E1 13557.49,E2 13557.49} C_VEL
LIN {X 0,Y 492.508,Z 1222.597,A -85,B 0,C 180,E1 13562.591,E2 13562.591} C_VEL
LIN {X 0,Y 487.787,Z 1248.338,A -85,B 0,C 180,E1 13568.17,E2 13568.17} C_VEL
LIN {X 0,Y 485.221,Z 1264.667,A -85,B 0,C 180,E1 13573.251,E2 13573.251} C_VEL
LIN {X 0,Y 484.674,Z 1269.33,A -85,B 0,C 180,E1 13575.119,E2 13575.119} C_VEL
LIN {X 0,Y 480.176,Z 1273.883,A -85,B 0,C 180,E1 13577.055,E2 13577.055} C_VEL
LIN {X 0,Y 475.873,Z 1277.696,A -85,B 0,C 180,E1 13579.047,E2 13579.047} C_VEL
LIN {X 0,Y 475.465,Z 1284.627,A -85,B 0,C 180,E1 13584.522,E2 13584.522} C_VEL
LIN {X 0,Y 475.534,Z 1287,A -85,B 0,C 180,E1 13589.993,E2 13589.993} C_VEL
LIN {X 0,Y 475.455,Z 1284.642,A -85,B 0,C 180,E1 13595.464,E2 13595.464} C_VEL
LIN {X 0,Y 475.917,Z 1277.658,A -85,B 0,C 180,E1 13600.974,E2 13600.974} C_VEL
LIN {X 0,Y 477.229,Z 1265.859,A -85,B 0,C 180,E1 13606.549,E2 13606.549} C_VEL
LIN {X 0,Y 479.202,Z 1252.49,A -85,B 0,C 180,E1 13610.691,E2 13610.691} C_VEL
LIN {X 0,Y 482.772,Z 1231.046,A -85,B 0,C 180,E1 13615.607,E2 13615.607} C_VEL
LIN {X 0,Y 488.019,Z 1203.943,A -85,B 0,C 180,E1 13620.457,E2 13620.457} C_VEL
LIN {X 0,Y 494.705,Z 1170.625,A -85,B 0,C 180,E1 13625.1,E2 13625.1} C_VEL
LIN {X 0,Y 502.845,Z 1130.819,A -85,B 0,C 180,E1 13629.477,E2 13629.477} C_VEL
LIN {X 0,Y 511.156,Z 1087.495,A -85,B 0,C 180,E1 13633.171,E2 13633.171} C_VEL
LIN {X 0,Y 519.947,Z 1038.79,A -85,B 0,C 180,E1 13636.392,E2 13636.392} C_VEL
LIN {X 0,Y 528.455,Z 984.463,A -85,B 0,C 180,E1 13639.048,E2 13639.048} C_VEL
LIN {X 0,Y 535.723,Z 931.471,A -85,B 0,C 180,E1 13640.891,E2 13640.891} C_VEL
LIN {X 0,Y 535.875,Z 924.708,A -85,B 0,C 180,E1 13641.142,E2 13641.142} C_VEL
LIN {X 0,Y 519.215,Z 880.618,A -85,B 0,C 180,E1 13645.007,E2 13645.007} C_VEL
LIN {X 0,Y 514.462,Z 865.743,A -85,B 0,C 180,E1 13647.025,E2 13647.025} C_VEL
LIN {X 0,Y 513.594,Z 861.431,A -85,B 0,C 180,E1 13648.024,E2 13648.024} C_VEL
LIN {X 0,Y 513.001,Z 862.239,A -85,B 0,C 180,E1 13648.939,E2 13648.939} C_VEL
LIN {X 0,Y 514.077,Z 871.284,A -85,B 0,C 180,E1 13650.991,E2 13650.991} C_VEL
LIN {X 0,Y 520.634,Z 896.86,A -85,B 0,C 180,E1 13654.615,E2 13654.615} C_VEL
LIN {X 0,Y 528.373,Z 928.454,A -85,B 0,C 180,E1 13658.49,E2 13658.49} C_VEL
LIN {X 0,Y 518.942,Z 969.225,A -85,B 0,C 180,E1 13661.539,E2 13661.539} C_VEL
LIN {X 0,Y 509.46,Z 1003.858,A -85,B 0,C 180,E1 13664.958,E2 13664.958} C_VEL
LIN {X 0,Y 499.877,Z 1036.339,A -85,B 0,C 180,E1 13669.11,E2 13669.11} C_VEL
LIN {X 0,Y 490.793,Z 1065.491,A -85,B 0,C 180,E1 13674.035,E2 13674.035} C_VEL
LIN {X 0,Y 484.141,Z 1088.334,A -85,B 0,C 180,E1 13679.127,E2 13679.127} C_VEL
LIN {X 0,Y 479.016,Z 1107.653,A -85,B 0,C 180,E1 13684.976,E2 13684.976} C_VEL
LIN {X 0,Y 476.236,Z 1123.871,A -85,B 0,C 180,E1 13691.901,E2 13691.901} C_VEL
LIN {X 0,Y 475.304,Z 1132.735,A -85,B 0,C 180,E1 13697.522,E2 13697.522} C_VEL
LIN {X 0,Y 474.616,Z 1136.538,A -85,B 0,C 180,E1 13702.609,E2 13702.609} C_VEL
LIN {X 0,Y 474.744,Z 1135.989,A -85,B 0,C 180,E1 13708.516,E2 13708.516} C_VEL
LIN {X 0,Y 475.545,Z 1131.325,A -85,B 0,C 180,E1 13713.513,E2 13713.513} C_VEL
LIN {X 0,Y 476.549,Z 1122.118,A -85,B 0,C 180,E1 13718.866,E2 13718.866} C_VEL
LIN {X 0,Y 479.147,Z 1106.203,A -85,B 0,C 180,E1 13725.262,E2 13725.262} C_VEL
LIN {X 0,Y 483.96,Z 1086.382,A -85,B 0,C 180,E1 13730.949,E2 13730.949} C_VEL
LIN {X 0,Y 490.734,Z 1061.456,A -85,B 0,C 180,E1 13736.235,E2 13736.235} C_VEL
LIN {X 0,Y 499.452,Z 1031.678,A -85,B 0,C 180,E1 13741.057,E2 13741.057} C_VEL
LIN {X 0,Y 509.276,Z 997.431,A -85,B 0,C 180,E1 13745.274,E2 13745.274} C_VEL
LIN {X 0,Y 519.466,Z 959.505,A -85,B 0,C 180,E1 13748.894,E2 13748.894} C_VEL
LIN {X 0,Y 527.32,Z 925.763,A -85,B 0,C 180,E1 13751.436,E2 13751.436} C_VEL
LIN {X 0,Y 516.482,Z 892.115,A -85,B 0,C 180,E1 13755.608,E2 13755.608} C_VEL
LIN {X 0,Y 502.647,Z 859.85,A -85,B 0,C 180,E1 13759.835,E2 13759.835} C_VEL
LIN {X 0,Y 485.817,Z 827.809,A -85,B 0,C 180,E1 13764.414,E2 13764.414} C_VEL
LIN {X 0,Y 476.983,Z 813.883,A -85,B 0,C 180,E1 13766.659,E2 13766.659} C_VEL
LIN {X 0,Y 475.287,Z 809.06,A -85,B 0,C 180,E1 13767.274,E2 13767.274} C_VEL
LIN {X 0,Y 475.344,Z 809.06,A -85,B 0,C 180,E1 13771.829,E2 13771.829} C_VEL
LIN {X 0,Y 475.071,Z 809.06,A -85,B 0,C 180,E1 13777.317,E2 13777.317} C_VEL
LIN {X 0,Y 474.838,Z 809.06,A -85,B 0,C 180,E1 13782.879,E2 13782.879} C_VEL
LIN {X 0,Y 474.591,Z 809.06,A -85,B 0,C 180,E1 13788.573,E2 13788.573} C_VEL
LIN {X 0,Y 474.293,Z 809.06,A -85,B 0,C 180,E1 13794.475,E2 13794.475} C_VEL
LIN {X 0,Y 474.157,Z 809.06,A -85,B 0,C 180,E1 13800.665,E2 13800.665} C_VEL
LIN {X 0,Y 474.003,Z 809.06,A -85,B 0,C 180,E1 13807.288,E2 13807.288} C_VEL
LIN {X 0,Y 473.904,Z 809.06,A -85,B 0,C 180,E1 13812.835,E2 13812.835} C_VEL
LIN {X 0,Y 473.853,Z 809.06,A -85,B 0,C 180,E1 13817.962,E2 13817.962} C_VEL
LIN {X 0,Y 473.954,Z 809.06,A -85,B 0,C 180,E1 13824.982,E2 13824.982} C_VEL
LIN {X 0,Y 474.23,Z 809.06,A -85,B 0,C 180,E1 13831.451,E2 13831.451} C_VEL
LIN {X 0,Y 474.405,Z 809.06,A -85,B 0,C 180,E1 13837.531,E2 13837.531} C_VEL
LIN {X 0,Y 474.634,Z 809.06,A -85,B 0,C 180,E1 13843.351,E2 13843.351} C_VEL
LIN {X 0,Y 474.921,Z 809.06,A -85,B 0,C 180,E1 13848.996,E2 13848.996} C_VEL
LIN {X 0,Y 475.189,Z 809.06,A -85,B 0,C 180,E1 13854.527,E2 13854.527} C_VEL
LIN {X 0,Y 475.572,Z 809.06,A -85,B 0,C 180,E1 13860.001,E2 13860.001} C_VEL
LIN {X 0,Y 475.228,Z 809.06,A -85,B 0,C 180,E1 13865.474,E2 13865.474} C_VEL
LIN {X 0,Y 474.926,Z 809.06,A -85,B 0,C 180,E1 13871.006,E2 13871.006} C_VEL
LIN {X 0,Y 474.585,Z 809.06,A -85,B 0,C 180,E1 13877.194,E2 13877.194} C_VEL
LIN {X 0,Y 474.286,Z 809.06,A -85,B 0,C 180,E1 13883.467,E2 13883.467} C_VEL
LIN {X 0,Y 474.327,Z 809.681,A -85,B 0,C 180,E1 13884.151,E2 13884.151} C_VEL
LIN {X 0,Y 476.975,Z 815.014,A -85,B 0,C 180,E1 13884.813,E2 13884.813} C_VEL
LIN {X 0,Y 499.607,Z 847.783,A -85,B 0,C 180,E1 13889.562,E2 13889.562} C_VEL
LIN {X 0,Y 525.224,Z 888.728,A -85,B 0,C 180,E1 13894.249,E2 13894.249} C_VEL
LIN {X 0,Y 544.204,Z 924.823,A -85,B 0,C 180,E1 13897.689,E2 13897.689} C_VEL
LIN {X 0,Y 545.427,Z 929.084,A -85,B 0,C 180,E1 13897.986,E2 13897.986} C_VEL
LIN {X 0,Y 538.175,Z 979.335,A -85,B 0,C 180,E1 13899.516,E2 13899.516} C_VEL
LIN {X 0,Y 529.584,Z 1027.52,A -85,B 0,C 180,E1 13901.735,E2 13901.735} C_VEL
LIN {X 0,Y 520.16,Z 1072.295,A -85,B 0,C 180,E1 13904.501,E2 13904.501} C_VEL
LIN {X 0,Y 509.5,Z 1117.35,A -85,B 0,C 180,E1 13908.188,E2 13908.188} C_VEL
LIN {X 0,Y 500.459,Z 1154.868,A -85,B 0,C 180,E1 13912.139,E2 13912.139} C_VEL
LIN {X 0,Y 491.67,Z 1191.58,A -85,B 0,C 180,E1 13917.067,E2 13917.067} C_VEL
LIN {X 0,Y 485.081,Z 1221.251,A -85,B 0,C 180,E1 13922.135,E2 13922.135} C_VEL
LIN {X 0,Y 480.091,Z 1247.025,A -85,B 0,C 180,E1 13927.801,E2 13927.801} C_VEL
LIN {X 0,Y 477.464,Z 1264.663,A -85,B 0,C 180,E1 13932.97,E2 13932.97} C_VEL
LIN {X 0,Y 476.018,Z 1276.071,A -85,B 0,C 180,E1 13938.085,E2 13938.085} C_VEL
LIN {X 0,Y 475.873,Z 1277.696,A -85,B 0,C 180,E1 13939.047,E2 13939.047} C_VEL
LIN {X 0,Y 471.706,Z 1280.946,A -85,B 0,C 180,E1 13941.069,E2 13941.069} C_VEL
LIN {X 0,Y 467.605,Z 1283.432,A -85,B 0,C 180,E1 13943.141,E2 13943.141} C_VEL
LIN {X 0,Y 467.515,Z 1286.663,A -85,B 0,C 180,E1 13948.14,E2 13948.14} C_VEL
LIN {X 0,Y 467.707,Z 1286.667,A -85,B 0,C 180,E1 13951.844,E2 13951.844} C_VEL
LIN {X 0,Y 467.684,Z 1282.919,A -85,B 0,C 180,E1 13957.418,E2 13957.418} C_VEL
LIN {X 0,Y 468.39,Z 1274.288,A -85,B 0,C 180,E1 13963.043,E2 13963.043} C_VEL
LIN {X 0,Y 469.627,Z 1263.559,A -85,B 0,C 180,E1 13967.3,E2 13967.3} C_VEL
LIN {X 0,Y 472.438,Z 1244.724,A -85,B 0,C 180,E1 13972.562,E2 13972.562} C_VEL
LIN {X 0,Y 476.699,Z 1221.392,A -85,B 0,C 180,E1 13977.534,E2 13977.534} C_VEL
LIN {X 0,Y 482.558,Z 1192.316,A -85,B 0,C 180,E1 13982.392,E2 13982.392} C_VEL
LIN {X 0,Y 489.732,Z 1158.34,A -85,B 0,C 180,E1 13986.859,E2 13986.859} C_VEL
LIN {X 0,Y 498.127,Z 1117.481,A -85,B 0,C 180,E1 13991.075,E2 13991.075} C_VEL
LIN {X 0,Y 506.899,Z 1073.928,A -85,B 0,C 180,E1 13994.59,E2 13994.59} C_VEL
LIN {X 0,Y 515.328,Z 1026.844,A -85,B 0,C 180,E1 13997.517,E2 13997.517} C_VEL
LIN {X 0,Y 523.359,Z 977.096,A -85,B 0,C 180,E1 13999.877,E2 13999.877} C_VEL
LIN {X 0,Y 529.808,Z 928.334,A -85,B 0,C 180,E1 14001.596,E2 14001.596} C_VEL
LIN {X 0,Y 515.207,Z 886.559,A -85,B 0,C 180,E1 14005.386,E2 14005.386} C_VEL
LIN {X 0,Y 511.52,Z 872.265,A -85,B 0,C 180,E1 14007.395,E2 14007.395} C_VEL
LIN {X 0,Y 511.061,Z 868.784,A -85,B 0,C 180,E1 14008.462,E2 14008.462} C_VEL
LIN {X 0,Y 510.462,Z 875.485,A -85,B 0,C 180,E1 14010.211,E2 14010.211} C_VEL
LIN {X 0,Y 514.445,Z 896.339,A -85,B 0,C 180,E1 14013.477,E2 14013.477} C_VEL
LIN {X 0,Y 522.752,Z 930.537,A -85,B 0,C 180,E1 14017.928,E2 14017.928} C_VEL
LIN {X 0,Y 513.055,Z 970.956,A -85,B 0,C 180,E1 14020.985,E2 14020.985} C_VEL
LIN {X 0,Y 502.985,Z 1006.456,A -85,B 0,C 180,E1 14024.537,E2 14024.537} C_VEL
LIN {X 0,Y 492.959,Z 1039.11,A -85,B 0,C 180,E1 14028.798,E2 14028.798} C_VEL
LIN {X 0,Y 483.372,Z 1068.784,A -85,B 0,C 180,E1 14033.943,E2 14033.943} C_VEL
LIN {X 0,Y 476.509,Z 1091.159,A -85,B 0,C 180,E1 14039.113,E2 14039.113} C_VEL
LIN {X 0,Y 471.33,Z 1110.165,A -85,B 0,C 180,E1 14045.057,E2 14045.057} C_VEL
LIN {X 0,Y 468.61,Z 1123.624,A -85,B 0,C 180,E1 14051.154,E2 14051.154} C_VEL
LIN {X 0,Y 467.49,Z 1132.193,A -85,B 0,C 180,E1 14056.911,E2 14056.911} C_VEL
LIN {X 0,Y 466.906,Z 1135.739,A -85,B 0,C 180,E1 14060.853,E2 14060.853} C_VEL
LIN {X 0,Y 466.7,Z 1136.704,A -85,B 0,C 180,E1 14066.953,E2 14066.953} C_VEL
LIN {X 0,Y 467.572,Z 1132.37,A -85,B 0,C 180,E1 14072.849,E2 14072.849} C_VEL
LIN {X 0,Y 468.866,Z 1122.255,A -85,B 0,C 180,E1 14079.346,E2 14079.346} C_VEL
LIN {X 0,Y 471.367,Z 1108.502,A -85,B 0,C 180,E1 14085.161,E2 14085.161} C_VEL
LIN {X 0,Y 476.2,Z 1089.109,A -85,B 0,C 180,E1 14090.913,E2 14090.913} C_VEL
LIN {X 0,Y 482.9,Z 1065.537,A -85,B 0,C 180,E1 14096.118,E2 14096.118} C_VEL
LIN {X 0,Y 492.31,Z 1034.266,A -85,B 0,C 180,E1 14101.328,E2 14101.328} C_VEL
LIN {X 0,Y 501.833,Z 1002.217,A -85,B 0,C 180,E1 14105.404,E2 14105.404} C_VEL
LIN {X 0,Y 512.574,Z 963.683,A -85,B 0,C 180,E1 14109.185,E2 14109.185} C_VEL
LIN {X 0,Y 520.893,Z 928.754,A -85,B 0,C 180,E1 14111.891,E2 14111.891} C_VEL
LIN {X 0,Y 510.506,Z 895.699,A -85,B 0,C 180,E1 14116.092,E2 14116.092} C_VEL
LIN {X 0,Y 496.362,Z 862.261,A -85,B 0,C 180,E1 14120.59,E2 14120.59} C_VEL
LIN {X 0,Y 479.793,Z 831.196,A -85,B 0,C 180,E1 14125.209,E2 14125.209} C_VEL
LIN {X 0,Y 469.494,Z 814.385,A -85,B 0,C 180,E1 14127.99,E2 14127.99} C_VEL
LIN {X 0,Y 467.446,Z 809.06,A -85,B 0,C 180,E1 14128.826,E2 14128.826} C_VEL
LIN {X 0,Y 467.325,Z 809.06,A -85,B 0,C 180,E1 14133.715,E2 14133.715} C_VEL
LIN {X 0,Y 467.086,Z 809.06,A -85,B 0,C 180,E1 14139.316,E2 14139.316} C_VEL
LIN {X 0,Y 466.839,Z 809.06,A -85,B 0,C 180,E1 14145.015,E2 14145.015} C_VEL
LIN {X 0,Y 466.533,Z 809.06,A -85,B 0,C 180,E1 14150.88,E2 14150.88} C_VEL
LIN {X 0,Y 466.328,Z 809.06,A -85,B 0,C 180,E1 14156.986,E2 14156.986} C_VEL
LIN {X 0,Y 466.125,Z 809.06,A -85,B 0,C 180,E1 14163.451,E2 14163.451} C_VEL
LIN {X 0,Y 465.971,Z 809.06,A -85,B 0,C 180,E1 14170.443,E2 14170.443} C_VEL
LIN {X 0,Y 465.986,Z 809.06,A -85,B 0,C 180,E1 14177.084,E2 14177.084} C_VEL
LIN {X 0,Y 465.926,Z 809.06,A -85,B 0,C 180,E1 14181.964,E2 14181.964} C_VEL
LIN {X 0,Y 466.12,Z 809.06,A -85,B 0,C 180,E1 14188.758,E2 14188.758} C_VEL
LIN {X 0,Y 466.392,Z 809.06,A -85,B 0,C 180,E1 14195.134,E2 14195.134} C_VEL
LIN {X 0,Y 466.633,Z 809.06,A -85,B 0,C 180,E1 14201.107,E2 14201.107} C_VEL
LIN {X 0,Y 466.845,Z 809.06,A -85,B 0,C 180,E1 14206.906,E2 14206.906} C_VEL
LIN {X 0,Y 467.168,Z 809.06,A -85,B 0,C 180,E1 14213.132,E2 14213.132} C_VEL
LIN {X 0,Y 467.474,Z 809.06,A -85,B 0,C 180,E1 14218.148,E2 14218.148} C_VEL
LIN {X 0,Y 467.397,Z 809.06,A -85,B 0,C 180,E1 14223.708,E2 14223.708} C_VEL
LIN {X 0,Y 467.108,Z 809.06,A -85,B 0,C 180,E1 14229.309,E2 14229.309} C_VEL
LIN {X 0,Y 466.779,Z 809.06,A -85,B 0,C 180,E1 14235.009,E2 14235.009} C_VEL
LIN {X 0,Y 466.514,Z 809.06,A -85,B 0,C 180,E1 14240.873,E2 14240.873} C_VEL
LIN {X 0,Y 466.442,Z 809.445,A -85,B 0,C 180,E1 14242.616,E2 14242.616} C_VEL
LIN {X 0,Y 468.81,Z 814.754,A -85,B 0,C 180,E1 14243.256,E2 14243.256} C_VEL
LIN {X 0,Y 471.372,Z 818.007,A -85,B 0,C 180,E1 14243.873,E2 14243.873} C_VEL
LIN {X 0,Y 495.98,Z 854.01,A -85,B 0,C 180,E1 14249.173,E2 14249.173} C_VEL
LIN {X 0,Y 520.303,Z 893.219,A -85,B 0,C 180,E1 14253.739,E2 14253.739} C_VEL
LIN {X 0,Y 539.059,Z 929.446,A -85,B 0,C 180,E1 14257.285,E2 14257.285} C_VEL
LIN {X 0,Y 539.439,Z 933.885,A -85,B 0,C 180,E1 14257.5,E2 14257.5} C_VEL
LIN {X 0,Y 532.108,Z 981.371,A -85,B 0,C 180,E1 14259.01,E2 14259.01} C_VEL
LIN {X 0,Y 523.052,Z 1030.057,A -85,B 0,C 180,E1 14261.303,E2 14261.303} C_VEL
LIN {X 0,Y 513.157,Z 1074.976,A -85,B 0,C 180,E1 14264.164,E2 14264.164} C_VEL
LIN {X 0,Y 502.126,Z 1119.91,A -85,B 0,C 180,E1 14267.934,E2 14267.934} C_VEL
LIN {X 0,Y 492.171,Z 1159.495,A -85,B 0,C 180,E1 14272.289,E2 14272.289} C_VEL
LIN {X 0,Y 483.63,Z 1193.889,A -85,B 0,C 180,E1 14277.088,E2 14277.088} C_VEL
LIN {X 0,Y 476.604,Z 1224.489,A -85,B 0,C 180,E1 14282.586,E2 14282.586} C_VEL
LIN {X 0,Y 472.139,Z 1247.512,A -85,B 0,C 180,E1 14287.87,E2 14287.87} C_VEL
LIN {X 0,Y 469.47,Z 1264.968,A -85,B 0,C 180,E1 14293.154,E2 14293.154} C_VEL
LIN {X 0,Y 468.155,Z 1276.068,A -85,B 0,C 180,E1 14297.882,E2 14297.882} C_VEL
LIN {X 0,Y 467.605,Z 1283.432,A -85,B 0,C 180,E1 14303.141,E2 14303.141} C_VEL
LIN {X 0,Y 463.524,Z 1285.3,A -85,B 0,C 180,E1 14305.22,E2 14305.22} C_VEL
LIN {X 0,Y 459.56,Z 1286.34,A -85,B 0,C 180,E1 14307.341,E2 14307.341} C_VEL
LIN {X 0,Y 459.799,Z 1286.667,A -85,B 0,C 180,E1 14311.876,E2 14311.876} C_VEL
LIN {X 0,Y 459.785,Z 1282.895,A -85,B 0,C 180,E1 14317.546,E2 14317.546} C_VEL
LIN {X 0,Y 460.459,Z 1274.257,A -85,B 0,C 180,E1 14322.79,E2 14322.79} C_VEL
LIN {X 0,Y 461.995,Z 1261.016,A -85,B 0,C 180,E1 14327.872,E2 14327.872} C_VEL
LIN {X 0,Y 465.036,Z 1241.861,A -85,B 0,C 180,E1 14333.194,E2 14333.194} C_VEL
LIN {X 0,Y 470.176,Z 1215.096,A -85,B 0,C 180,E1 14338.812,E2 14338.812} C_VEL
LIN {X 0,Y 476.528,Z 1184.763,A -85,B 0,C 180,E1 14343.696,E2 14343.696} C_VEL
LIN {X 0,Y 484.489,Z 1147.588,A -85,B 0,C 180,E1 14348.385,E2 14348.385} C_VEL
LIN {X 0,Y 493.027,Z 1107.281,A -85,B 0,C 180,E1 14352.387,E2 14352.387} C_VEL
LIN {X 0,Y 502.453,Z 1060.277,A -85,B 0,C 180,E1 14355.985,E2 14355.985} C_VEL
LIN {X 0,Y 511.45,Z 1011.214,A -85,B 0,C 180,E1 14358.862,E2 14358.862} C_VEL
LIN {X 0,Y 520.277,Z 956.715,A -85,B 0,C 180,E1 14361.215,E2 14361.215} C_VEL
LIN {X 0,Y 523.547,Z 931.207,A -85,B 0,C 180,E1 14362.126,E2 14362.126} C_VEL
LIN {X 0,Y 511.745,Z 894.043,A -85,B 0,C 180,E1 14365.604,E2 14365.604} C_VEL
LIN {X 0,Y 508.849,Z 879.852,A -85,B 0,C 180,E1 14367.578,E2 14367.578} C_VEL
LIN {X 0,Y 508.795,Z 876.542,A -85,B 0,C 180,E1 14368.339,E2 14368.339} C_VEL
LIN {X 0,Y 507.548,Z 882.94,A -85,B 0,C 180,E1 14370.022,E2 14370.022} C_VEL
LIN {X 0,Y 510.1,Z 902.369,A -85,B 0,C 180,E1 14373.163,E2 14373.163} C_VEL
LIN {X 0,Y 516.796,Z 934.596,A -85,B 0,C 180,E1 14377.482,E2 14377.482} C_VEL
LIN {X 0,Y 506.618,Z 975.093,A -85,B 0,C 180,E1 14380.621,E2 14380.621} C_VEL
LIN {X 0,Y 495.998,Z 1010.889,A -85,B 0,C 180,E1 14384.313,E2 14384.313} C_VEL
LIN {X 0,Y 485.967,Z 1042.116,A -85,B 0,C 180,E1 14388.51,E2 14388.51} C_VEL
LIN {X 0,Y 476.292,Z 1070.962,A -85,B 0,C 180,E1 14393.624,E2 14393.624} C_VEL
LIN {X 0,Y 469.023,Z 1093.554,A -85,B 0,C 180,E1 14398.979,E2 14398.979} C_VEL
LIN {X 0,Y 463.613,Z 1112.658,A -85,B 0,C 180,E1 14405.134,E2 14405.134} C_VEL
LIN {X 0,Y 460.841,Z 1125.692,A -85,B 0,C 180,E1 14411.345,E2 14411.345} C_VEL
LIN {X 0,Y 459.58,Z 1133.4,A -85,B 0,C 180,E1 14417.211,E2 14417.211} C_VEL
LIN {X 0,Y 458.751,Z 1136.915,A -85,B 0,C 180,E1 14423.28,E2 14423.28} C_VEL
LIN {X 0,Y 458.806,Z 1136.671,A -85,B 0,C 180,E1 14427.455,E2 14427.455} C_VEL
LIN {X 0,Y 459.612,Z 1133.364,A -85,B 0,C 180,E1 14432.571,E2 14432.571} C_VEL
LIN {X 0,Y 460.848,Z 1125.317,A -85,B 0,C 180,E1 14438.531,E2 14438.531} C_VEL
LIN {X 0,Y 463.036,Z 1113.197,A -85,B 0,C 180,E1 14444.127,E2 14444.127} C_VEL
LIN {X 0,Y 467.306,Z 1096.164,A -85,B 0,C 180,E1 14449.716,E2 14449.716} C_VEL
LIN {X 0,Y 474.158,Z 1072.109,A -85,B 0,C 180,E1 14455.459,E2 14455.459} C_VEL
LIN {X 0,Y 482.586,Z 1045.158,A -85,B 0,C 180,E1 14460.349,E2 14460.349} C_VEL
LIN {X 0,Y 492.949,Z 1011.621,A -85,B 0,C 180,E1 14464.966,E2 14464.966} C_VEL
LIN {X 0,Y 503.537,Z 975.629,A -85,B 0,C 180,E1 14468.794,E2 14468.794} C_VEL
LIN {X 0,Y 514.582,Z 932.062,A -85,B 0,C 180,E1 14472.311,E2 14472.311} C_VEL
LIN {X 0,Y 505.014,Z 900.777,A -85,B 0,C 180,E1 14476.379,E2 14476.379} C_VEL
LIN {X 0,Y 491.504,Z 867.856,A -85,B 0,C 180,E1 14480.903,E2 14480.903} C_VEL
LIN {X 0,Y 475.801,Z 837.651,A -85,B 0,C 180,E1 14485.485,E2 14485.485} C_VEL
LIN {X 0,Y 462.124,Z 814.851,A -85,B 0,C 180,E1 14489.364,E2 14489.364} C_VEL
LIN {X 0,Y 459.721,Z 809.686,A -85,B 0,C 180,E1 14490.125,E2 14490.125} C_VEL
LIN {X 0,Y 459.388,Z 809.06,A -85,B 0,C 180,E1 14495.671,E2 14495.671} C_VEL
